PROPERTY P_pParentMzTool : POINTER TO FB_MzBase
GET
END_GET
END_PROPERTY

PROPERTY P_pPiece : POINTER TO FB_PieceBase
GET
P_pPiece := pPiece;
END_GET
SET
pPiece := P_pPiece;
END_SET
END_PROPERTY

PROPERTY P_pXDrive : POINTER TO FB_XYDriveBase
GET
P_pXDrive := pXDrive;
END_GET
END_PROPERTY

PROPERTY P_pYDrive : POINTER TO FB_XYDriveBase
GET
P_pYDrive := pYDrive;
END_GET
END_PROPERTY

PROPERTY P_rToolRadius : REAL
GET
END_GET
END_PROPERTY

PROPERTY P_stAbsPosPhys : ST_3DPoint
GET
END_GET
END_PROPERTY

PROPERTY P_stAbsPosTotal : ST_3DPoint
GET
P_stAbsPosTotal := P_stAbsPosPhys;
END_GET
END_PROPERTY

PROPERTY P_stCurrentPosPhys : ST_3DPoint
GET
END_GET
END_PROPERTY

PROPERTY P_stCurrentPosTotal : ST_3DPoint
GET
P_stCurrentPosTotal := P_stCurrentPosPhys;
END_GET
END_PROPERTY

PROPERTY P_stError : ST_Error
GET
P_stError := stError;
END_GET
END_PROPERTY

PROPERTY P_stOffset : ST_3DPoint
GET
P_stOffset := stOffset;
END_GET
SET
stOffset := P_stOffset;
END_SET
END_PROPERTY

PROPERTY P_stRelPos : ST_3DPoint
GET
P_stRelPos := stRelPos;
END_GET
SET
stRelPos := P_stRelPos;
END_SET
END_PROPERTY

END_FUNCTION_BLOCK

// ---- Objects/FB_SlotList.TcPOU
FUNCTION_BLOCK FB_SlotList
VAR_INPUT
END_VAR
VAR_OUTPUT
END_VAR
VAR
	pHead	: POINTER TO ST_POINTER2;
	pTail	: POINTER TO ST_POINTER2;
	pCurrent: POINTER TO ST_POINTER2;
	nCount	: UINT;
END_VAR

PROPERTY P_nCount : UINT
GET
P_nCount := nCount;
END_GET
END_PROPERTY

METHOD M_GetAtIndex : POINTER TO FB_Slot
VAR_INPUT
	nIndex : UINT;
END_VAR

VAR
	i : UINT;
	pItem : POINTER TO ST_POINTER2;
END_VAR
//mit Index ist die fortlaufende Nummer eines Slots in der Liste gemeint
IF nIndex > 0 AND nIndex <= nCount THEN
	pItem := pHead;
	FOR i := 1 TO nIndex - 1 BY 1 DO
		pItem := pItem^.pNext;
	END_FOR
	M_GetAtIndex := pItem^.pContent;
END_IF
END_METHOD

METHOD M_GetAtNr : POINTER TO FB_Slot
VAR_INPUT
	nNr	: UINT;
END_VAR

VAR
	pPointer : POINTER TO ST_POINTER2;
	pSlot: POINTER TO FB_Slot; 
END_VAR
//Gibt Slot anhand der SlotNr zurück
pPointer := pHead;
WHILE pPointer > 0 DO
	pSlot := pPointer^.pContent;
	IF pSlot^.P_nNr = nNr THEN
		EXIT;
	ELSE
		pSlot := 0;
	END_IF
	pPointer := pPointer^.pNext;
END_WHILE

IF pSlot > 0 THEN
	M_GetAtNr := pSlot;
END_IF
END_METHOD

METHOD M_SetCurrentToHead : BOOL
VAR_INPUT
END_VAR
pCurrent := pHead;
END_METHOD

METHOD M_Add : ERRORID
VAR_INPUT
	pSlot : POINTER TO FB_Slot;
END_VAR

VAR
	pNew : POINTER TO ST_POINTER2;
END_VAR
pNew := pHead;
WHILE pNew > 0 DO
	IF pNew^.pContent = pSlot THEN
		M_Add := 43434;
		RETURN;
	END_IF
	pNew := pNew^.pNext;
END_WHILE

pNew := __NEW(ST_Pointer2);
MEMSET(pNew,0,SIZEOF(ST_POINTER2));
pNew^.pContent := pSlot;
IF pHead = 0 THEN
	pHead := pTail := pNew;
ELSE
	pNew^.pPrev := pTail; 
	pTail^.pNext := pNew;
	pTail := pNew;
END_IF
nCount := nCount + 1;
END_METHOD

METHOD M_Reset
VAR_INPUT
END_VAR

VAR
	pDelete : POINTER TO ST_Pointer2;
	pNext	: POINTER TO ST_Pointer2;
	pSlot	: POINTER TO FB_SLOT;
END_VAR
pDelete := pHead;
WHILE  pDelete > 0 DO
	pNext := pDelete^.pNext;
	pSlot := pDelete^.pContent; 
	IF pSlot > 0 THEN
		__DELETE(pSlot);
	END_IF
	__DELETE(pDelete);
	pDelete := pNext;
END_WHILE
pHead := 0;
pTail := 0;
pCurrent := 0;
nCount := 0;
END_METHOD

METHOD M_GetNext : POINTER TO FB_Slot
VAR_INPUT
END_VAR

VAR
	pSlot : POINTER TO FB_Slot;
END_VAR
IF pCurrent > 0 THEN
	pSlot := pCurrent^.pContent;
	IF pSlot > 0 THEN
		M_GetNext := pSlot;
	END_IF
	pCurrent := pCurrent^.pNext;
END_IF
END_METHOD

END_FUNCTION_BLOCK

// ---- Objects/Targets/Passive/FB_Workplate.TcPOU
FUNCTION_BLOCK FB_Workplate EXTENDS FB_SlotTarget
VAR_INPUT
END_VAR
VAR_OUTPUT
END_VAR
VAR
	rCollHeight			: REAL;
	bCalcCollHeight		: BOOL;
	iter				: FB_ObjCollectIteratorDeep;
	pTarget				: POINTER TO FB_TargetBase;
	stAbsPosCenter		: ST_3DPoint;
	fbRectangle			: FB_Rectangle;
	nParentSlotNr		: UINT;		//Workplate befindet sich zwar an keinem Slot, aber virtuell in der GUI (am Root)
END_VAR

IF bCalcCollHeight THEN
	bCalcCollHeight := FALSE;
	fbRectangle(X1:=0.0, Y1:=0.0, X2:=stDimension.Width, Y2:=stDimension.Depth);
	pTarget := M_GetHighestTarget(fbRectAngle,0.0);
	IF pTarget > 0 THEN
		IF pTarget^.P_rAbsFreeHeight > P_rAbsFreeHeight THEN
			rCollHeight := pTarget^.P_rAbsFreeHeight + 1000.0;
		ELSE
			rCollHeight := P_rAbsFreeHeight + 1000.0;
		END_IF
	ELSE
		rCollHeight := P_rAbsFreeHeight + 1000.0;
	END_IF
END_IF

METHOD FB_init : BOOL
VAR_INPUT
	bInitRetains : BOOL; // if TRUE, the retain variables are initialized (warm start / cold start)
	bInCopyCode : BOOL;  // if TRUE, the instance afterwards gets moved into the copy code (online change)
END_VAR
eObjectType := E_ObjectType.OBJECTTYPE_Workplate;
eObjectGroup := E_ObjectGroup.OBJECTGROUP_Target;
END_METHOD

METHOD M_AddChild : ERRORID
VAR_INPUT
	pObject : POINTER TO FB_Object;
	nSlotNr	: UINT;
	nIndex 	: INT;
END_VAR
//Kann alle Targets aufnehmen
IF pObject > 0 THEN
	IF pObject^.M_bIsGroup(E_ObjectGroup.OBJECTGROUP_Target) THEN
		M_AddChild := SUPER^.M_AddChild(pObject,nSlotNr,nIndex);
	ELSE
		M_AddChild := E_ErrorIdObjMgmt.ERRORID_InvalidParentObject;
	END_IF
ELSE
	M_AddChild := E_ErrorIdObjMgmt.ERRORID_InvalidParentObject;
END_IF
END_METHOD

METHOD M_ClearAllProps
VAR_INPUT
	bIgnoreParent : BOOL; //Es wird das gesamte OD gelöscht. -> Zeiger auf Parent nicht mehr gültig!
END_VAR
SUPER^.M_ClearAllProps(bIgnoreParent);
rCollHeight := 0;
END_METHOD

METHOD M_GetAllProps : ERRORID
VAR_INPUT
	refCmdData : REFERENCE TO  ST_CmdData;
END_VAR
SUPER^.M_GetAllProps(refCmdData);

refCmdData.n32Data[1] := nParentSlotNr;
END_METHOD

METHOD M_SetAllProps : ERRORID
VAR_INPUT
	refCmdData : REFERENCE TO  ST_CmdData;
END_VAR
M_SetAllProps := SUPER^.M_SetAllProps(refCmdData);
IF M_SetAllProps > 0 THEN
	RETURN;
END_IF

nParentSlotNr := DINT_TO_UINT(refCmdData.n32Data[1]);
END_METHOD

PROPERTY P_bCalcCollisHeight : BOOL
SET
bCalcCollHeight := P_bCalcCollisHeight;
END_SET
END_PROPERTY

PROPERTY P_nParentSlotNr : UINT
GET
P_nParentSlotNr := nParentSlotNr;
END_GET
END_PROPERTY

PROPERTY P_rCollHeight : REAL
GET
P_rCollHeight := rCollHeight;
END_GET
SET
rCollHeight := P_rCollHeight;
END_SET
END_PROPERTY

END_FUNCTION_BLOCK

// ---- Objects/Targets/Passive/FB_SlotTarget.TcPOU
FUNCTION_BLOCK FB_SlotTarget EXTENDS FB_TargetBase IMPLEMENTS I_SlotTarget
VAR_INPUT
END_VAR
VAR_OUTPUT
END_VAR
VAR
	fbSlotList			: FB_SlotList;
	nNumberOfSlots		: UINT;
	nFirstSlotPropIndex	: UINT;	//erster Index für Slots (benötigt in M_SetSingleProps)
	nLastSlotPropIndex	: UINT;	//letzte Index für Slots (benötigt in M_SetSingleProps)
END_VAR

SUPER^();

METHOD M_AddChild : ERRORID
VAR_INPUT
	pObject : POINTER TO FB_Object;
	nSlotNr	: UINT;
	nIndex 	: INT;
END_VAR

VAR
	pSlot : POINTER TO FB_Slot;
END_VAR
//In den abgeleiteten Tool-FBs wird überprüft, ob das entsprechende Objekt als Child tauglich ist
IF pObject > 0 THEN
	IF nSlotNr > 0 THEN
		pSlot := fbSlotList.M_GetAtNr(nSlotNr);
		IF pSlot > 0 THEN
			IF pSlot^.P_pChild = 0 THEN
				//Object darf selber noch an keinem Parent hängen
				IF pObject^.P_pParentObject = 0 THEN
					pSlot^.P_pChild := pObject;
					pObject^.P_pObjCollectNode := pObjCollectNode^.nodes.M_AddNewNode(pObject,nIndex);
					pObject^.M_UpdateParent();
				ELSE
					M_AddChild := E_ErrorIdObjMgmt.ERRORID_ObjectAlreadyOnAnotherParent;
				END_IF
			ELSE //Slot bereits belegt
				M_AddChild := E_ErrorIdObjMgmt.ERRORID_SlotIsAlreadyOccupied;
			END_IF		
		ELSE
			M_AddChild := E_ErrorIdObjMgmt.ERRORID_InvalidSlotNumber;			
		END_IF	
	ELSE
		M_AddChild := SUPER^.M_AddChild(pObject,nSlotNr,nIndex);
	END_IF
ELSE
	M_AddChild := E_ErrorIdObjMgmt.ERRORID_InvalidParentObject;
END_IF
END_METHOD

METHOD M_ApplyPos : ERRORID
VAR_INPUT
	eTargetRef 		: E_TargetRef;
	nPointSlotNr	: UINT;
	stPos 			: ST_3DPoint;
	bXPos			: BOOL;
	bYPos			: BOOL;
	bZPos			: BOOL;	
END_VAR

VAR
	stAbsPos		: ST_3DPoint;
	pSlot			: POINTER TO FB_Slot;
END_VAR
IF eTargetRef = E_TargetRef.TARGETREF_Slot THEN
	stAbsPos := P_stAbsPosLB;
	pSlot := M_GetSlot(nPointSlotNr);
	IF pSlot > 0 THEN
		IF bXPos THEN
			pSlot^.P_rRelPosX := stPos.X - stAbsPos.X;
		END_IF
		IF bYPos THEN
			pSlot^.P_rRelPosY := stPos.Y - stAbsPos.Y;
		END_IF
		IF bZPos THEN
			pSlot^.P_rRelPosZ := stPos.Z - stAbsPos.Z;
			P_pWorkplate^.P_bCalcCollisHeight := TRUE;
		END_IF
	ELSE
		M_ApplyPos := E_ErrorIdCmd.ERRORID_InvalidTargetSlot;
	END_IF
ELSE
	M_ApplyPos := SUPER^.M_ApplyPos(eTargetRef, nPointSlotNr, stPos,bXPos, bYPos, bZPos);	
END_IF
END_METHOD

METHOD M_ClearAllProps
VAR_INPUT
	bIgnoreParent : BOOL; //Es wird das gesamte OD gelöscht. -> Zeiger auf Parent nicht mehr gültig!
END_VAR
fbSlotList.M_Reset();
SUPER^.M_ClearAllProps(bIgnoreParent);
END_METHOD

METHOD M_GetAbsPos : ST_3DPoint
VAR_INPUT
	pChildPos	: POINTER TO ST_3DPoint;
	eTargetRef 	: E_TargetRef;
	nParam1		: UINT;
 	nParam2		: UINT;
	nParam3		: USINT;
	nParam4		: USINT;
	nZLevel		: USINT;
END_VAR
VAR_OUTPUT
	nErrorId 	: ERRORID;
	lrAngle		: LREAL;
END_VAR
VAR
	stLocPos : ST_3DPoint;
	pSlot : POINTER TO FB_Slot;
END_VAR
IF eTargetRef = E_TargetRef.TARGETREF_Slot THEN
	//Slotnummer checken
	pSlot := M_GetSlot(nParam1);
	IF pSlot > 0 THEN
		stLocPos := F_Add3DPoints(pSlot^.P_stRelPos,stRelPos);
		stLocPos.Z := stLocPos.Z + stDimension.Height;
		//kann es mal sein, dass hier das ParentTarget = 0 ist?
		//ja -> bei der Workplate
		IF pChildPos > 0 THEN
			stLocPos := F_Add3DPoints(stLocPos,pChildPos^);
		END_IF
		IF pParentTarget > 0 THEN
			IF pParentSlot > 0 THEN
				M_GetAbsPos := pParentTarget^.M_GetAbsPos(pChildPos := ADR(stLocPos), eTargetRef:= E_TargetRef.TARGETREF_Slot,
															nParam1:= pParentSlot^.P_nNr,
															nParam2:= 0, nParam3:= 0, nParam4:= 0,nZLevel:= 0, lrAngle=> lrAngle,
															nErrorId=> nErrorId);		
			ELSE
				M_GetAbsPos := pParentTarget^.M_GetAbsPos(pChildPos := ADR(stLocPos), eTargetRef:= E_TargetRef.TARGETREF_LeftBottom,
																nParam1:= 0,
																nParam2:= 0, nParam3:= 0, nParam4:= 0, nZLevel:= 0,
																lrAngle => lrAngle, nErrorId=> nErrorId);
			END_IF
		ELSE
			M_GetAbsPos := stLocPos;
		END_IF		
	ELSE
		nErrorId := E_ErrorIdCmd.ERRORID_InvalidTargetSlot;
	END_IF
	
ELSE
	M_GetAbsPos := SUPER^.M_GetAbsPos(pChildPos := pChildPos, eTargetRef:= eTargetRef,
													nParam1:= nParam1,
													nParam2:= nParam2, nParam3:= nParam3, nParam4:= 0, nZLevel:= nZLevel,
													lrAngle => lrAngle, nErrorId=> nErrorId);	
END_IF
END_METHOD

METHOD M_GetAllProps : ERRORID
VAR_INPUT
	refCmdData : REFERENCE TO  ST_CmdData;
END_VAR

VAR
	i : UINT;
	pSlot		: POINTER TO FB_Slot;
	pPieceSlot	: POINTER TO FB_PieceSlot;
END_VAR
SUPER^.M_GetAllProps(refCmdData);

nCurrentPropIndex := nCurrentPropIndex + 1;

refCmdData.n32Data[nCurrentPropIndex] := fbSlotList.P_nCount;

fbSlotList.M_SetCurrentToHead();

IF (eObjectGroup AND E_ObjectGroup.OBJECTGROUP_Rack) = E_ObjectGroup.OBJECTGROUP_Rack THEN
	FOR i := 1 TO fbSlotList.P_nCount BY 1 DO
		pPieceSlot := fbSlotList.M_GetNext();
		IF pPieceSlot > 0 THEN
			nCurrentPropIndex := nCurrentPropIndex + 1;
			refCmdData.n32Data[nCurrentPropIndex] := pPieceSlot^.P_nNr;
			nCurrentPropIndex := nCurrentPropIndex + 1;
			refCmdData.n32Data[nCurrentPropIndex] := REAL_TO_DINT(pPieceSlot^.P_rRelPosX);
			nCurrentPropIndex := nCurrentPropIndex + 1;
			refCmdData.n32Data[nCurrentPropIndex] := REAL_TO_DINT(pPieceSlot^.P_rRelPosY);
			nCurrentPropIndex := nCurrentPropIndex + 1;
			refCmdData.n32Data[nCurrentPropIndex] := REAL_TO_DINT(pPieceSlot^.P_rRelPosZ);
			nCurrentPropIndex := nCurrentPropIndex + 1;
			refCmdData.n32Data[nCurrentPropIndex] := REAL_TO_DINT(pPieceSlot^.P_rDepth);
		END_IF		
	END_FOR	
ELSE
	FOR i := 1 TO fbSlotList.P_nCount BY 1 DO
		pSlot := fbSlotList.M_GetNext();
		IF pSlot > 0 THEN
			nCurrentPropIndex := nCurrentPropIndex + 1;
			refCmdData.n32Data[nCurrentPropIndex] := pSlot^.P_nNr;
			nCurrentPropIndex := nCurrentPropIndex + 1;
			refCmdData.n32Data[nCurrentPropIndex] := REAL_TO_DINT(pSlot^.P_rRelPosX);
			nCurrentPropIndex := nCurrentPropIndex + 1;
			refCmdData.n32Data[nCurrentPropIndex] := REAL_TO_DINT(pSlot^.P_rRelPosY);
			nCurrentPropIndex := nCurrentPropIndex + 1;
			refCmdData.n32Data[nCurrentPropIndex] := REAL_TO_DINT(pSlot^.P_rRelPosZ);
		END_IF		
	END_FOR	
END_IF
END_METHOD

METHOD M_GetSlot : POINTER TO FB_Slot
VAR_INPUT
	nSlotNr : UINT;
END_VAR
M_GetSlot := fbSlotList.M_GetAtNr(nSlotNr);
END_METHOD

METHOD M_GetSlotFromChild : POINTER TO FB_Slot
VAR_INPUT
	pObject : POINTER TO FB_Object;
END_VAR

VAR
	pSlot : POINTER TO FB_Slot;
END_VAR
//Die SlotList iterieren und vergleichen ob Objekte übereinstimmen
fbSlotList.M_SetCurrentToHead();
REPEAT
	pSlot := fbSlotList.M_GetNext();
	IF pSlot > 0 THEN
		IF pSlot^.P_pChild = pObject THEN
			M_GetSlotFromChild := pSlot;
			EXIT;
		END_IF
	END_IF
UNTIL pSlot = 0
END_REPEAT
END_METHOD

METHOD M_SetAllProps : ERRORID
VAR_INPUT
	refCmdData : REFERENCE TO  ST_CmdData;
END_VAR

VAR
	i : UINT;
	pSlot 		: POINTER TO FB_Slot;
	pPieceSlot	: POINTER TO FB_PieceSlot;
END_VAR
M_SetAllProps := SUPER^.M_SetAllProps(refCmdData);

IF M_SetAllProps > 0 THEN
	RETURN;
END_IF

//Slots parametrieren
nCurrentPropIndex := nCurrentPropIndex + 1;
nFirstSlotPropIndex := nCurrentPropIndex;
nNumberOfSlots := DINT_TO_UINT(refCmdData.n32Data[nCurrentPropIndex]);

//Falls SlotList noch nicht existiert, dann neue erstellen
IF fbSlotList.P_nCount = 0 THEN
	FOR i:= 1 TO nNumberOfSlots BY 1 DO
		IF (eObjectGroup AND E_ObjectGroup.OBJECTGROUP_Rack) = E_ObjectGroup.OBJECTGROUP_Rack THEN
			pPieceSlot := __NEW(FB_PieceSlot(pOwner := THIS));
			pSlot := pPieceSlot;
		ELSE
			pSlot := __NEW(FB_Slot(pOwner := THIS));
		END_IF
		
		fbSlotList.M_Add(pSlot);
		nCurrentPropIndex := nCurrentPropIndex + 1;
		pSlot^.P_nNr := DINT_TO_USINT(refCmdData.n32Data[nCurrentPropIndex]);
		nCurrentPropIndex := nCurrentPropIndex + 1;
		pSlot^.P_rRelPosX := DINT_TO_REAL(refCmdData.n32Data[nCurrentPropIndex]);
		nCurrentPropIndex := nCurrentPropIndex + 1;
		pSlot^.P_rRelPosY := DINT_TO_REAL(refCmdData.n32Data[nCurrentPropIndex]);
		nCurrentPropIndex := nCurrentPropIndex + 1;
		pSlot^.P_rRelPosZ := DINT_TO_REAL(refCmdData.n32Data[nCurrentPropIndex]);
		
		IF (eObjectGroup AND E_ObjectGroup.OBJECTGROUP_Rack) = E_ObjectGroup.OBJECTGROUP_Rack THEN
			nCurrentPropIndex := nCurrentPropIndex + 1;
			pPieceSlot^.P_rDepth := DINT_TO_REAL(refCmdData.n32Data[nCurrentPropIndex]);
		END_IF
	END_FOR
ELSE
	IF nNumberOfSlots <> fbSlotList.P_nCount THEN	//Anzahl der Slots dürfen sich nicht ändern
		M_SetAllProps := E_ErrorIdObjMgmt.ERRORID_ChangeNoOfSlotsNotAllowed;
		RETURN;		
	END_IF

	FOR i:= 1 TO nNumberOfSlots BY 1 DO
		nCurrentPropIndex := nCurrentPropIndex + 1;
		IF (eObjectGroup AND E_ObjectGroup.OBJECTGROUP_Rack) = E_ObjectGroup.OBJECTGROUP_Rack THEN
			pPieceSlot := fbSlotList.M_GetAtNr(DINT_TO_USINT(refCmdData.n32Data[nCurrentPropIndex]));
			IF pPieceSlot > 0 THEN
				nCurrentPropIndex := nCurrentPropIndex + 1;
				pPieceSlot^.P_rRelPosX := DINT_TO_REAL(refCmdData.n32Data[nCurrentPropIndex]);
				nCurrentPropIndex := nCurrentPropIndex + 1;
				pPieceSlot^.P_rRelPosY := DINT_TO_REAL(refCmdData.n32Data[nCurrentPropIndex]);
				nCurrentPropIndex := nCurrentPropIndex + 1;
				pPieceSlot^.P_rRelPosZ := DINT_TO_REAL(refCmdData.n32Data[nCurrentPropIndex]);
				nCurrentPropIndex := nCurrentPropIndex + 1;
				pPieceSlot^.P_rDepth := DINT_TO_REAL(refCmdData.n32Data[nCurrentPropIndex]);
			ELSE
				M_SetAllProps := 222;
				RETURN;
			END_IF 
		ELSE
			pSlot := fbSlotList.M_GetAtNr(DINT_TO_USINT(refCmdData.n32Data[nCurrentPropIndex]));
			IF pSlot > 0 THEN
				nCurrentPropIndex := nCurrentPropIndex + 1;
				pSlot^.P_rRelPosX := DINT_TO_REAL(refCmdData.n32Data[nCurrentPropIndex]);
				nCurrentPropIndex := nCurrentPropIndex + 1;
				pSlot^.P_rRelPosY := DINT_TO_REAL(refCmdData.n32Data[nCurrentPropIndex]);
				nCurrentPropIndex := nCurrentPropIndex + 1;
				pSlot^.P_rRelPosZ := DINT_TO_REAL(refCmdData.n32Data[nCurrentPropIndex]);
			ELSE
				M_SetAllProps := 222;
				RETURN;
			END_IF	
		END_IF
	END_FOR
END_IF
nLastSlotPropIndex := nCurrentPropIndex;
nNoOfProps := nCurrentPropIndex + 1;
END_METHOD

METHOD M_SetSingleProp : ERRORID
VAR_INPUT
	refCmdData : REFERENCE TO  ST_CmdData;
END_VAR

VAR
	nSlotNr		: UINT;
	nIndex		: UINT;
	pSlot		: POINTER TO FB_Slot;
	pPieceSlot	: POINTER TO FB_PieceSlot;
END_VAR
//Handelt es sich bei dem PropNr um eine SlotPropNr?
IF refCmdData.aHeader[1] >= nFirstSlotPropIndex AND refCmdData.aHeader[1] <= nLastSlotPropIndex THEN
	nIndex := (refCmdData.aHeader[1]- nFirstSlotPropIndex);
	//Beachten normale Slots oder PieceSlots
	IF (eObjectGroup AND E_ObjectGroup.OBJECTGROUP_Rack) = E_ObjectGroup.OBJECTGROUP_Rack THEN //PieceSlots
		IF nIndex MOD 5 = 0 THEN
			nSlotNr := nIndex / 5;
		ELSE
			nSlotNr := nIndex / 5 + 1;
		END_IF
		pPieceSlot := fbSlotList.M_GetAtNr(nSlotNr);
		IF pPieceSlot > 0 THEN
			nIndex := nIndex - ((nSlotNr - 1)* 5);
			CASE nIndex OF
				2:	pPieceSlot^.P_rRelPosX := DINT_TO_REAL(refCmdData.n32Data[0]);
				
				3:	pPieceSlot^.P_rRelPosY := DINT_TO_REAL(refCmdData.n32Data[0]);
				
				4:	pPieceSlot^.P_rRelPosZ := DINT_TO_REAL(refCmdData.n32Data[0]);
					P_pWorkplate^.P_bCalcCollisHeight := TRUE;
				
				5:	pPieceSlot^.P_rDepth := DINT_TO_REAL(refCmdData.n32Data[0]);
			END_CASE
		END_IF
	ELSE //normale Slots
		IF nIndex MOD 4 = 0 THEN
			nSlotNr := nIndex / 4;
		ELSE
			nSlotNr := nIndex / 4 + 1;
		END_IF
		pSlot := fbSlotList.M_GetAtNr(nSlotNr);
		IF pSlot > 0 THEN
			nIndex := nIndex - ((nSlotNr - 1)* 4);
			CASE nIndex OF
				2:	pSlot^.P_rRelPosX := DINT_TO_REAL(refCmdData.n32Data[0]);
				
				3:	pSlot^.P_rRelPosY := DINT_TO_REAL(refCmdData.n32Data[0]);
				
				4:	pSlot^.P_rRelPosZ := DINT_TO_REAL(refCmdData.n32Data[0]);
					P_pWorkplate^.P_bCalcCollisHeight := TRUE;
			END_CASE
		END_IF	
	END_IF
ELSE
	M_SetSingleProp := SUPER^.M_SetSingleProp(refCmdData);
END_IF
END_METHOD

END_FUNCTION_BLOCK

// ---- Functions/F_Add3DPoints.TcPOU
FUNCTION F_Add3DPoints : ST_3DPoint
VAR_INPUT
	stPoint1	: ST_3DPoint;
	stPoint2	: ST_3DPoint;
END_VAR
VAR
	_stPoint	: ST_3DPoint;
END_VAR

_stPoint.X := stPoint1.X + stPoint2.X;
_stPoint.Y := stPoint1.Y + stPoint2.Y;
_stPoint.Z := stPoint1.Z + stPoint2.Z;
F_Add3DPoints := _stPoint;

END_FUNCTION

// ---- Objects/FB_PieceSlot.TcPOU
{attribute 'enable_dynamic_creation'}
FUNCTION_BLOCK FB_PieceSlot EXTENDS FB_Slot
VAR_INPUT
END_VAR
VAR_OUTPUT
END_VAR
VAR
	rDepth	 : REAL;
END_VAR

PROPERTY P_rDepth : REAL
GET
P_rDepth := rDepth;
END_GET
SET
rDepth := P_rDepth;
END_SET
END_PROPERTY

PROPERTY P_pPiece : POINTER TO FB_PieceBase
GET
IF pChild > 0 THEN
	P_pPiece := pChild;
END_IF
END_GET
SET
IF P_pPiece > 0 THEN
	pChild := P_pPiece;
ELSE
	pChild := 0;	
END_IF
END_SET
END_PROPERTY

END_FUNCTION_BLOCK

// ---- Objects/Pieces/FB_PieceBase.TcPOU
FUNCTION_BLOCK FB_PieceBase EXTENDS FB_Object
VAR_INPUT
END_VAR
VAR_OUTPUT
	bUsingPiece			: BOOL;	
END_VAR
VAR
	pParentObject		: POINTER TO FB_Object;
	stDimension			: ST_3DDimension;
	rSlotDiameter		: REAL;
	stOffset			: ST_3DPoint;	//Offset
	rZOverlapTool		: REAL;
	rZOverlapSlot		: REAL;
	rMeasureDistance	: REAL;
	rDockOffset			: REAL;
	nCurrentPropIndex	: USINT;
	nSpecPropIndex		: USINT;			//erster Index für Specialproperties
	bIgnoreOffset		: BOOL;
END_VAR

METHOD M_UpdateParent
VAR_INPUT
END_VAR
IF pObjCollectNode > 0 AND_THEN pObjCollectNode^.pOwnerColl > 0 THEN
	pParentObject := pObjCollectNode^.pOwnerColl^.pOwnerNode^.P_pObject;
ELSE
	pParentObject := 0;
END_IF

IF pParentObject > 0 THEN
	pParentSlot := pParentObject^.M_GetSlotFromChild(THIS);
ELSE
	pParentSlot := 0;
END_IF
END_METHOD

METHOD M_GetPropCheckSum : UINT
VAR_INPUT
END_VAR

VAR
	stData 		: ST_CmdData;
END_VAR
M_GetAllProps(stData);
wChecksum := F_DATA_TO_CRC16_CCITT(ADR(stData.n32Data[0]),nNoOfProps * 4,16#FFFF);
M_GetPropCheckSum := wChecksum;
END_METHOD

PROPERTY P_stDimension : ST_3DDimension
GET
P_stDimension := stDimension;
END_GET
END_PROPERTY

PROPERTY P_rDockOffset : REAL
GET
P_rDockOffset := rDockOffset;
END_GET
END_PROPERTY

{attribute 'object_name' := 'M_CheckProps'}
METHOD M_CheckProps : ERRORID
END_METHOD

PROPERTY P_rZOverlapSlot : REAL
GET
P_rZOverlapSlot := rZOverlapSlot;
END_GET
END_PROPERTY

PROPERTY P_pLatestChild : POINTER TO FB_PieceBase
GET
P_pLatestChild := THIS;
END_GET
END_PROPERTY

PROPERTY P_rZOverlapTool : REAL
GET
P_rZOverlapTool := rZOverlapTool;
END_GET
END_PROPERTY

PROPERTY P_stOffset : ST_3DPoint
GET
P_stOffset := stOffset;
END_GET
SET
stOffset := P_stOffset;
END_SET
END_PROPERTY

{attribute 'object_name' := 'M_ClearAllProps'}
METHOD M_ClearAllProps

VAR_INPUT
	bIgnoreParent : BOOL; //Es wird das gesamte OD gelöscht. -> Zeiger auf Parent nicht mehr gültig!
END_VAR
IF NOT bIgnoreParent THEN
	IF pParentSlot > 0 THEN
		pParentSlot^.P_pChild := 0;
	END_IF	
END_IF
nObjectID := 0;
pParentObject := 0;
pParentSlot := 0;
pObjCollectNode := 0;
END_METHOD

METHOD M_GetRelPosTopCenter : ST_3DPoint
VAR_INPUT
END_VAR
VAR
	stPosTemp : ST_3DPoint;
	pPieceSlot : POINTER TO FB_PieceSlot;
END_VAR
IF pParentObject > 0 THEN
	IF pParentObject^.M_bIsGroup(E_ObjectGroup.OBJECTGROUP_Target) THEN
		IF pParentSlot > 0 THEN
			pPieceSlot := pParentSlot;
			stPosTemp := pPieceSlot^.P_stRelPos;
			//Wenn OverlapSlot > SlotTiefe, dann sitzt Piece auf dem Grund des Slots auf
			IF rZOverlapSlot > pPieceSlot^.rDepth THEN
				stPosTemp.Z := stPosTemp.Z - pPieceSlot^.rDepth + stDimension.Height;
			ELSE
				stPosTemp.Z := stPosTemp.Z - rZOverlapSlot + stDimension.Height;
			END_IF
			IF bIgnoreOffset THEN
				M_GetRelPosTopCenter := stPosTemp;
			ELSE
				M_GetRelPosTopCenter := F_Add3DPoints(stPosTemp,stOffset);	
			END_IF
		END_IF
	END_IF
END_IF
END_METHOD

{attribute 'object_name' := 'M_SetSingleProp'}
METHOD M_SetSingleProp : ERRORID
VAR_INPUT
	refCmdData	: REFERENCE TO ST_CmdData;
END_VAR
CASE refCmdData.aHeader[1] OF
	0,1:
		M_SetSingleProp := E_ErrorIdCmd.ERRORID_InvalidProperty;
	2:	stDimension.Width := DINT_TO_REAL(refCmdData.n32Data[0]);
	3:	stDimension.Depth := DINT_TO_REAL(refCmdData.n32Data[0]);
	4:	stDimension.Height := DINT_TO_REAL(refCmdData.n32Data[0]);
	5:	rSlotDiameter := DINT_TO_REAL(refCmdData.n32Data[0]);
	6:	rZOverlapTool := DINT_TO_REAL(refCmdData.n32Data[0]);
	7:	rZOverlapSlot := DINT_TO_REAL(refCmdData.n32Data[0]);
	8:	stOffset.X := DINT_TO_REAL(refCmdData.n32Data[0]);
	9:	stOffset.Y := DINT_TO_REAL(refCmdData.n32Data[0]);
	10:	stOffset.Z := DINT_TO_REAL(refCmdData.n32Data[0]);
	11: rMeasureDistance := DINT_TO_REAL(refCmdData.n32Data[0]);
	12:	rDockOffset := DINT_TO_REAL(refCmdData.n32Data[0]);
END_CASE
END_METHOD

METHOD M_ClearOffset
VAR_INPUT
END_VAR
stOffset.X := 0.0;
stOffset.Y := 0.0;
stOffset.Z := 0.0;
END_METHOD

PROPERTY P_rMeasureDistance : REAL
GET
P_rMeasureDistance := rMeasureDistance;
END_GET
END_PROPERTY

{attribute 'object_name' := 'M_GetAllProps'}
METHOD M_GetAllProps : ERRORID
VAR_INPUT
	refCmdData	: REFERENCE TO ST_CmdData;
END_VAR
refCmdData.aHeader[0] := nObjectID;
refCmdData.aHeader[1] := eObjectType;
refCmdData.aHeader[2] := 0;

IF pParentObject > 0 THEN
	refCmdData.n32Data[0] := pParentObject^.P_nObjectID;
ELSE
	refCmdData.n32Data[0] := 0;
END_IF

IF pParentSlot > 0 THEN
	refCmdData.n32Data[1] := pParentSlot^.nNr;
ELSE
	refCmdData.n32Data[1] := 0;
END_IF

//Dimensionen lesen
refCmdData.n32Data[2] := REAL_TO_DINT(stDimension.Width);
refCmdData.n32Data[3] := REAL_TO_DINT(stDimension.Depth);
refCmdData.n32Data[4] := REAL_TO_DINT(stDimension.Height);
refCmdData.n32Data[5] := REAL_TO_DINT(rSlotDiameter);
refCmdData.n32Data[6] := REAL_TO_DINT(rZOverlapTool);
refCmdData.n32Data[7] := REAL_TO_DINT(rZOverlapSlot);
refCmdData.n32Data[8] := REAL_TO_DINT(stOffset.X);
refCmdData.n32Data[9] := REAL_TO_DINT(stOffset.Y);
refCmdData.n32Data[10] := REAL_TO_DINT(stOffset.Z);
refCmdData.n32Data[11] := REAL_TO_DINT(rMeasureDistance);
refCmdData.n32Data[12] := REAL_TO_DINT(rDockOffset);
nCurrentPropIndex := 12;
END_METHOD

METHOD M_AddChild : ERRORID
VAR_INPUT
	pObject	: POINTER TO FB_Object;
	nSlotNr	: UINT;
	nIndex 	: INT;
END_VAR
//Pieces könnnen keine Childs aufnehmen
M_AddChild := E_ErrorIdObjMgmt.ERRORID_ObjectCanNotTakeChilds;
END_METHOD

{attribute 'object_name' := 'M_SetAllProps'}
METHOD M_SetAllProps : ERRORID
VAR_INPUT
	refCmdData	: REFERENCE TO ST_CmdData;
END_VAR
IF fbObjectDirectory.M_GetObjPointer(DINT_TO_UINT(refCmdData.n32Data[0])) = 0 THEN
	M_SetAllProps := E_ErrorIdObjMgmt.ERRORID_InvalidParentObject;
	RETURN;
END_IF

//ParentSlot unterschiedlich?

(*IF pParentSlot = 0 THEN
	M_SetAllProps := M_SetParent(aI_Object[refCmdData.n32Data[0]],DINT_TO_UINT(refCmdData.n32Data[1]));
ELSE
	IF pParentSlot^.P_nNr <> DINT_TO_UINT(refCmdData.n32Data[1]) THEN
		M_SetAllProps := M_SetParent(aI_Object[refCmdData.n32Data[0]],DINT_TO_UINT(refCmdData.n32Data[1]));
	END_IF
END_IF

IF M_SetAllProps > 0 THEN
	RETURN;
END_IF*)

//Dimensionen setzen
stDimension.Width := DINT_TO_REAL(refCmdData.n32Data[2]);
stDimension.Depth := DINT_TO_REAL(refCmdData.n32Data[3]);
stDimension.Height := DINT_TO_REAL(refCmdData.n32Data[4]);
rSlotDiameter := DINT_TO_REAL(refCmdData.n32Data[5]);
rZOverlapTool := DINT_TO_REAL(refCmdData.n32Data[6]);
rZOverlapSlot := DINT_TO_REAL(refCmdData.n32Data[7]);
stOffset.X := DINT_TO_REAL(refCmdData.n32Data[8]);
stOffset.Y := DINT_TO_REAL(refCmdData.n32Data[9]);
stOffset.Z := DINT_TO_REAL(refCmdData.n32Data[10]);
rMeasureDistance := DINT_TO_REAL(refCmdData.n32Data[11]);
rDockOffset := DINT_TO_REAL(refCmdData.n32Data[12]);
nCurrentPropIndex := 12;
nNoOfProps := nCurrentPropIndex + 1;
END_METHOD

PROPERTY P_nCntSlots : UINT
GET
END_GET
END_PROPERTY

PROPERTY P_bIgnoreOffset : BOOL
SET
bIgnoreOffset := P_bIgnoreOffset;
END_SET
GET
P_bIgnoreOffset := bIgnoreOffset;
END_GET
END_PROPERTY

END_FUNCTION_BLOCK

// ---- DUTs/Structs/FB_Rectangle.TcPOU
FUNCTION_BLOCK FB_Rectangle
VAR_INPUT
	X1,Y1,X2,Y2 : REAL;	
END_VAR
VAR_OUTPUT
END_VAR
VAR
END_VAR

PROPERTY P_LineLeft : ST_Line
GET
P_LineLeft.X1 := X1;
P_LineLeft.Y1 := Y1;
P_LineLeft.X2 := X1;
P_LineLeft.Y2 := Y2;
END_GET
END_PROPERTY

PROPERTY P_LineRight : ST_Line
GET
P_LineRight.X1 := X2;
P_LineRight.Y1 := Y1;
P_LineRight.X2 := X2;
P_LineRight.Y2 := Y2;
END_GET
END_PROPERTY

METHOD M_Clear
VAR_INPUT
END_VAR
X1 := 0;
Y1 := 0;
X2 := 0;
Y2 := 0;
END_METHOD

PROPERTY P_LineTop : ST_Line
GET
P_LineTop.X1 := X1;
P_LineTop.Y1 := Y2;
P_LineTop.X2 := X2;
P_LineTop.Y2 := Y2;
END_GET
END_PROPERTY

PROPERTY P_LineBottom : ST_Line
GET
P_LineBottom.X1 := X1;
P_LineBottom.Y1 := Y1;
P_LineBottom.X2 := X2;
P_LineBottom.Y2 := Y1;
END_GET
END_PROPERTY

END_FUNCTION_BLOCK

// ---- Hardware/MultiZ/FB_ZM_Home.TcPOU
FUNCTION_BLOCK FB_ZM_Home
VAR_INPUT
	bExecute		: BOOL;
	pFbZAxisRef		: POINTER TO FB_ZAxisRef;
	bMoveToHome		: BOOL;
END_VAR
VAR_OUTPUT
	bBusy		: BOOL;
	bError		: BOOL;
	nErrorId	: ERRORID;
END_VAR
VAR
	fbSdoWrite	: FB_SDO_WRITE;
	nState		: USINT;
	timeOut		: TON;
	bTest		: BOOL;
	tTime		: TIME;
	nErrorState : USINT;
END_VAR

IF bExecute THEN
	IF pFbZAxisRef = 0 THEN
		RETURN;
	END_IF
	
	//Fehler-Simualation
	(*IF pFbZAxisRef^.nChannel = 4 THEN
		bBusy := FALSE;
		bError := TRUE;
		nState := 99;	//go in errorstate
		RETURN;
	END_IF*)
	
	IF pFbZAxisRef^.stInput.nStatus.3 THEN //Error
		pFbZAxisRef^.stStatus.bError := TRUE;
		pFbZAxisRef^.stStatus.bIsMoving := FALSE;
		pFbZAxisRef^.stStatus.bIsHoming := FALSE;
		pFbZAxisRef^.stOutput.nMode := 0;
		pFbZAxisRef^.stOutput.nCtrl := 0;
		nErrorID := F_MultiZError_TO_ErrorId(pFbZAxisRef^.stInput.nError);
		timeOut(IN:= FALSE);
		bBusy := FALSE;
		bError := TRUE;
		nState := 99;	//go in errorstate
		RETURN;
	END_IF
	
	timeOut();
	IF timeOut.Q THEN
		tTime := timeOut.ET;
		nErrorState := nState;
		timeOut(IN:= FALSE);
		pFbZAxisRef^.stStatus.bError := TRUE;
		pFbZAxisRef^.stStatus.bIsMoving := FALSE;
		pFbZAxisRef^.stStatus.bIsHoming := FALSE;
		pFbZAxisRef^.stOutput.nMode := 0;
		pFbZAxisRef^.stOutput.nCtrl := 0;
		CASE nState OF
			0:	//Timeout reset error
				nErrorId := E_ErrorIdMultiZ.ERRORID_ToResetErr;
			3,6: //Timeout wait for setpointacknowledge
				nErrorId := E_ErrorIdMultiZ.ERRORID_ToWaitSetPointAck;
				bTest := TRUE;
			4: //Timeout wait for targetreached
				nErrorId := E_ErrorIdMultiZ.ERRORID_ToWaitTrgtReached;
		ELSE
			nErrorId := E_ErrorIdMultiZ.ERRORID_UnknownError;	
		END_CASE
		bBusy := FALSE;
		bError := TRUE;
		nState := 99;	//go in errorstate
		RETURN;
	END_IF
	
	CASE nState OF
		0:	bBusy := TRUE;
			pFbZAxisRef^.stStatus.bError := FALSE;
			pFbZAxisRef^.stStatus.bIsHomed := FALSE;
			pFbZAxisRef^.stStatus.bIsHoming := TRUE;
			
			//Das zurücksetzen von Fehlern sollte ausschließlich im FB_MultiZRef stattfinden!!!
			//Hier nur abfragen, ob "pFbZAxisRef^.stStatus.bError" und dann in Error gehen	
			IF pFbZAxisRef^.stInput.nStatus.3 THEN //Error
				pFbZAxisRef^.stOutput.nCtrl := 8;	//Error zurücksetzen
				pFbZAxisRef^.stOutput.nVelo := 0;	//Geschwindigkeit auf 0 setzen
				timeOut(IN:= TRUE, PT:=T#1000MS);	//Timer für Timeout starten
			ELSE
				//Mode of Operation setzen
				IF pFbZAxisRef^.P_bInvertInitDir THEN
					pFbZAxisRef^.stOutput.nMode := 7;
				ELSE
					pFbZAxisRef^.stOutput.nMode := 6;
					pFbZAxisRef^.stOutput.nVelo := 50000;
				END_IF
				
				fbSdoWrite(sADSNetID:= pFbZAxisRef^.pMultiZRef^.P_sAdsNetId, nPortNr:= pFbZAxisRef^.pMultiZRef^.P_nAdsPort,
							nIndex:= cRefPos.nIndex, nSubIndex:= pFbZAxisRef^.nChannel, 
							nDataLength:= cRefPos.nLength, nData:= REAL_TO_DINT(pFbZAxisRef^.P_rRefPos) , bExecute:= TRUE);
				nState := 1;
				timeOut(IN:= FALSE);
			END_IF
			
		1:	//Geschwindigkeit setzen
			fbSdoWrite();
			IF NOT fbSdoWrite.bBusy THEN
				IF fbSdoWrite.bError THEN
					nErrorId := fbSdoWrite.nAdsErrorId;
					bBusy := FALSE;
					bError := TRUE;
					nState := 99;	//go in errorstate
				ELSE
					nState := 200;	
				END_IF
				fbSdoWrite(bExecute:= FALSE);
			END_IF
			
		200:
			nState := 201;
			
		201:
			nState := 2;
						
		2:	//Fahrauftrag starten
			pFbZAxisRef^.stOutput.nCtrl := 1;
			pFbZAxisRef^.stStatus.bIsMoving := TRUE;
			timeOut(IN:= TRUE, PT:=T#2000MS);	//Timer für Timeout starten
			nState := 3;
	
		3:	//SetpointAcknowledge?
			IF pFbZAxisRef^.stInput.nStatus.1 THEN
				pFbZAxisRef^.stOutput.nCtrl := 0;	//Fahrauftrag zurücksetzen
				timeOut(IN:= FALSE);
				nState := 4;
			END_IF
			
		4:	//TargetReached?
			IF pFbZAxisRef^.stInput.nStatus.0 THEN
				pFbZAxisRef^.stStatus.bIsMoving := FALSE;	
				pFbZAxisRef^.stOutput.nMode := 1;		//in Positioniermodus umschalten
				timeOut(IN:= FALSE);
				IF bMoveToHome THEN
					pFbZAxisRef^.P_rAbsTargetPos := pFbZAxisRef^.P_rHomePos;
					nState := 5;
				ELSE
					nState := 8;
				END_IF
			ELSE
				timeOut(IN:= TRUE, PT:=T#5S);	//Timer für Timeout starten
			END_IF
			
		5:	//auf HomePos fahren
			pFbZAxisRef^.stOutput.nCtrl := 1;
			pFbZAxisRef^.stStatus.bIsMoving := TRUE;
			timeOut(IN:= TRUE, PT:=T#500MS);	//Timer für Timeout starten
			nState := 6;
			
		6:	//SetpointAcknowledge?
			IF pFbZAxisRef^.stInput.nStatus.1 THEN
				pFbZAxisRef^.stOutput.nCtrl := 0;	//Fahrauftrag zurücksetzen
				timeOut(IN:= FALSE);
				nState := 7;
			END_IF			
			
		7:	//TargetReached?
			IF pFbZAxisRef^.stInput.nStatus.0 THEN
				pFbZAxisRef^.stStatus.bIsMoving := FALSE;
				timeOut(IN:= FALSE);
				nState := 8;
			ELSE
				timeOut(IN:= TRUE, PT:=T#3S);	//Timer für Timeout starten
			END_IF	
		
		8:	IF pFbZAxisRef^.stInput.nStatus.3 THEN		//Error ist in Achse aufgetreten
				pFbZAxisRef^.stStatus.bError := TRUE;
				pFbZAxisRef^.stStatus.bIsMoving := FALSE;
				pFbZAxisRef^.stStatus.bIsHoming := FALSE;
				nErrorID := F_MultiZError_TO_ErrorId(pFbZAxisRef^.stInput.nError);
				bBusy := FALSE;
				bError := TRUE;
				nState := 99;	//go in errorstate
				RETURN;
			ELSE
				pFbZAxisRef^.stStatus.bIsHomed := pFbZAxisRef^.stInput.nStatus.6;
				pFbZAxisRef^.stStatus.bIsHoming := FALSE;
				bBusy := FALSE;
				nState := 9;
			END_IF
	END_CASE
ELSE
	bMoveToHome := FALSE;
	bError := FALSE;
	nErrorId := 0;
	nState := 0;
	timeOut(IN:= FALSE);
	IF pFbZAxisRef > 0 THEN
		pFbZAxisRef^.stStatus.bIsHoming := FALSE;
		pFbZAxisRef^.stOutput.nCtrl := 0;	//Fahrauftrag zurücksetzen (notwendig bei Cancel)	
		IF pFbZAxisRef^.stOutput.nMode = 6 THEN
			pFbZAxisRef^.stOutput.nMode := 0;
		END_IF
	END_IF
	bBusy := FALSE;
END_IF

END_FUNCTION_BLOCK

// ---- Hardware/MultiZ/FB_ZM_Move.TcPOU
FUNCTION_BLOCK FB_ZM_Move
VAR_INPUT
	bExecute		: BOOL;
	rPosition		: REAL;	//Zielposition bzw. Distance bei relativer Fahrt
	rSpeed			: REAL;	//Geschwindigkeit
	eMoveMode		: E_MoveMode;
	pfbZAxisRef		: POINTER TO FB_ZAxisRef;
END_VAR

VAR_OUTPUT
	bBusy			: BOOL;
	bCommandAborted	: BOOL;
	bError			: BOOL;
	nErrorID		: ERRORID;
END_VAR

VAR
	nState				: USINT;
	rCurrentPosition	: REAL;
	tWaitForTrgtReached	: TIME;
	timeOut				: TON;
	fbSdoRead			: FB_SDO_READ;
END_VAR

IF bExecute THEN
	IF pfbZAxisRef = 0 THEN
		nErrorId := E_ErrorIdMultiZ.ERRORID_InvalidZChannel;
		bBusy := FALSE;
		bError := TRUE;
		nState := 99;
		RETURN;
	END_IF
	
	//Wird Achse momentan von anderem Movebaustein genutzt?
	IF (pfbZAxisRef^.pCurrentFb > 0) AND (pfbZAxisRef^.pCurrentFb <> THIS) THEN //wird von anderem FB genutzt
		RETURN;
	END_IF
	
	IF pFbZAxisRef^.stInput.nStatus.3 THEN //Error
		pFbZAxisRef^.stStatus.bError := TRUE;
		pFbZAxisRef^.stOutput.nMode := 0;
		pFbZAxisRef^.stOutput.nCtrl := 0;
		timeOut(IN:= FALSE);
		nErrorID := F_MultiZError_TO_ErrorId(pFbZAxisRef^.stInput.nError);
		bBusy := FALSE;
		bError := TRUE;
		nState := 99;
		RETURN;
	END_IF
	
	IF pFbZAxisRef^.stStatus.bError THEN
		nErrorID := F_MultiZError_TO_ErrorId(pFbZAxisRef^.stInput.nError);
		bBusy := FALSE;
		bError := TRUE;
		nState := 99;
		RETURN;
	END_IF

	//Wenn durch anderen FB Achse gestoppt, dann abbrechen
	IF pFbZAxisRef^.stStatus.bCmdAborted THEN	//Muss noch irgendwo gesetzt werden!!!!
		bCommandAborted := TRUE;
		bBusy := FALSE;
	END_IF
	
	IF timeOut.Q THEN
		timeOut(IN:= FALSE);
		bError := TRUE;
		bBusy := FALSE;
		pFbZAxisRef^.stStatus.bError := TRUE;
		pFbZAxisRef^.stOutput.nCtrl.1 := TRUE;	//Stopbit setzen
		
		CASE nState OF
			2: //Timeout wait for setpointacknowledge
				nErrorId := E_ErrorIdMultiZ.ERRORID_ToWaitSetPointAck;
			3: //Timeout wait for targetreached
				nErrorId := E_ErrorIdMultiZ.ERRORID_ToWaitTrgtReached;
		ELSE
			nErrorId := E_ErrorIdMultiZ.ERRORID_UnknownError;	
		END_CASE
		nState := 99;
		RETURN;
	END_IF		
	
	CASE nState OF
		0:	bBusy := TRUE;
			//Wenn Achse schon aktiv, warten bis wieder frei
			(*IF pstMultiZRef^.stZAxisStatus[nChannel].bHasJob THEN
				RETURN;
			END_IF*)
			pfbZAxisRef^.pCurrentFb := THIS; 
		
			//Geschwindigkeit innerhalb zulässiger Grenzen?
			IF rSpeed <= 0.0 OR rSpeed > pFbZAxisRef^.P_rMaxSpeed THEN
				nErrorID := E_ErrorIdCmd.ERRORID_VelocityOutOfRange;
				bBusy := FALSE;
				bError := TRUE;
				nState := 99;
				RETURN;
			END_IF
			
			pFbZAxisRef^.stStatus.bIsMoving := TRUE;
			pFbZAxisRef^.stStatus.bHasJob := TRUE;
			
			//Aktuelle Position holen
			rCurrentPosition := pFbZAxisRef^.P_rCurrentPos;

			//Targetposition innerhalb zulässiger Grenzen?
			CASE eMoveMode OF
				E_MoveMode.MODE_Relative,E_MoveMode.MODE_Measure:
					IF (rCurrentPosition + rPosition) < pFbZAxisRef^.P_rMinPos OR (rCurrentPosition + rPosition) > pFbZAxisRef^.P_rMaxPos THEN
						nErrorID := E_ErrorIdCmd.ERRORID_TargetPosOutOfRangeZ;
						bError := TRUE;
						bBusy := FALSE;
						nState := 99;
					ELSE
						//Timeout-Zeit für Wait for Targetreached berechnen
						IF eMoveMode = E_MoveMode.MODE_Measure THEN
							//Measure hat fixe Speed "15000"
							tWaitForTrgtReached := REAL_TO_TIME(ABS(rPosition) / 15000 * 1000 + 2000);
						ELSE
							tWaitForTrgtReached := REAL_TO_TIME(ABS(rPosition) / rSpeed * 1000.0 + 2000.0);
						END_IF
					END_IF				

				E_MoveMode.MODE_AbsWithOffset,E_MoveMode.MODE_AbsNoneOffset,E_MoveMode.MODE_Free,E_MoveMode.MODE_Home:
					IF eMoveMode = E_MoveMode.MODE_Home THEN
						rPosition := pFbZAxisRef^.P_rHomePos;
					END_IF
					
					IF rPosition < pFbZAxisRef^.P_rMinPos OR rPosition > pFbZAxisRef^.P_rMaxPos THEN
						nErrorID := E_ErrorIdCmd.ERRORID_TargetPosOutOfRangeZ;
						bError := TRUE;
						bBusy := FALSE;
						nState := 99;
					ELSE
						//Timeout-Zeit für Wait for Targetreached berechnen
						tWaitForTrgtReached := REAL_TO_TIME(ABS(rCurrentPosition - rPosition) / rSpeed * 1000.0 + 2000.0);
					END_IF				
			END_CASE
			
			IF NOT bError THEN
				//Betriebsart Positionsmodus und TargetPos setzen
				IF eMoveMode = E_MoveMode.MODE_Measure THEN
					pFbZAxisRef^.stOutput.nMode := 5;  //Measure
					//Zielposition setzen
					pFbZAxisRef^.P_rRelTargetPos := rPosition;
				ELSIF eMoveMode = E_MoveMode.MODE_Relative THEN
					pFbZAxisRef^.stOutput.nMode := 1;  //Positioniermodus
					//Zielposition setzen
					pFbZAxisRef^.P_rRelTargetPos := rPosition;
				ELSE
					pFbZAxisRef^.stOutput.nMode := 1;
					//Zielposition setzen
					pFbZAxisRef^.P_rAbsTargetPos := rPosition;
				END_IF
				//Geschwindigkeit setzen
				pFbZAxisRef^.stOutput.nVelo := REAL_TO_DINT(rSpeed);
				nState := 1;
			END_IF

		1:	//Fahrauftrag starten
			IF eMoveMode = E_MoveMode.MODE_Relative THEN	//Relativ
				pFbZAxisRef^.stOutput.nCtrl := 5;
			ELSE
				pFbZAxisRef^.stOutput.nCtrl := 1;	
			END_IF
			nState := 2;
	
		2:	//SetpointAcknowledge?
			IF pFbZAxisRef^.stInput.nStatus.1 THEN
				pFbZAxisRef^.stOutput.nCtrl.0 := FALSE;	//Fahrauftrag zurücksetzen
				timeOut(IN:= FALSE);
				nState := 3;
			ELSE
				timeOut(IN:= TRUE, PT:=T#1200MS);	//Timer für Timeout starten
			END_IF
			
		3:	//TargetReached?
			//IF pFbZAxisRef^.stInput.nStatus.0 THEN
			IF pFbZAxisRef^.stInput.nStatus = 193 THEN
				timeOut(IN:= FALSE);
				IF eMoveMode = E_MoveMode.MODE_Measure THEN
					nState := 4;
				ELSE
					bBusy := FALSE;	
				END_IF
			ELSE
				timeOut(IN:= TRUE, PT:= tWaitForTrgtReached);	//Timer für Timeout starten
			END_IF
		
		4:	//wenn "MODE_Measure", dann ZOffset holen
			fbSdoRead(sADSNetID:= pFbZAxisRef^.pMultiZRef^.P_sAdsNetId,	nPortNr:= pFbZAxisRef^.pMultiZRef^.P_nAdsPort,
					nIndex:= cZSensOffset.nIndex, nSubIndex:= pFbZAxisRef^.nChannel, nDataLength:= cZSensOffset.nLength, bExecute:= TRUE);
			IF NOT fbSdoRead.bBusy THEN
				IF fbSdoRead.bError THEN
					bError := TRUE;
					nState := 99;
				ELSE
					pFbZAxisRef^.P_nZSensorID := fbSdoRead.nData;
				END_IF
				fbSdoRead(bExecute:= FALSE);
				bBusy := FALSE;
			END_IF
	END_CASE
ELSE
	bBusy := FALSE;
	nState := 0;
	bError := FALSE;
	nErrorID := 0;
	timeOut(IN:= FALSE);
	IF pfbZAxisRef^.pCurrentFb > 0 THEN
		IF pfbZAxisRef^.pCurrentFb = THIS THEN
			pfbZAxisRef^.pCurrentFb := 0;
			pFbZAxisRef^.stStatus.bCmdAborted := FALSE;
			pFbZAxisRef^.stOutput.nMode := 0;
			pFbZAxisRef^.stStatus.bHasJob := FALSE;
			pFbZAxisRef^.stStatus.bIsMoving := FALSE;		
		END_IF		
	END_IF
END_IF

END_FUNCTION_BLOCK

// ---- Hardware/MultiZ/FB_ZM_Stop.TcPOU
FUNCTION_BLOCK FB_ZM_Stop
VAR_INPUT
	bExecute		: BOOL;
	pFbZAxisRef		: POINTER TO FB_ZAxisRef;
END_VAR

VAR_OUTPUT
	bBusy			: BOOL;
	bError			: BOOL;
	nErrorID		: ERRORID;
END_VAR

VAR
	nState				: USINT;
	timeOut				: TON;
	nCurrentPosition	: REAL;
	//bFlagGetPosition 	: BOOL := TRUE;
	//fbMultiZReadSdoVar	: FB_MultiZReadSdoVar;
END_VAR

IF bExecute THEN
	IF pFbZAxisRef = 0 THEN
		nErrorId := E_ErrorIdMultiZ.ERRORID_InvalidZChannel;
		bError := TRUE;
		nState := 99;	//go in errorstate		
		RETURN;
	END_IF
	
	IF pFbZAxisRef^.stInput.nStatus.3 THEN //Error
		pFbZAxisRef^.stStatus.bError := TRUE;
		pFbZAxisRef^.stOutput.nMode := 0;
		pFbZAxisRef^.stOutput.nCtrl := 0;
		timeOut(IN:= FALSE);
		nErrorID := F_MultiZError_TO_ErrorId(pFbZAxisRef^.stInput.nError);
		bBusy := FALSE;
		bError := TRUE;
		nState := 99;	//go in errorstate
		RETURN;
	END_IF

	IF timeOut.Q THEN
		timeOut(IN:= FALSE);
		bError := TRUE;
		bBusy := FALSE;
		pFbZAxisRef^.stStatus.bError := TRUE;
		pFbZAxisRef^.stOutput.nMode := 0;
		pFbZAxisRef^.stOutput.nCtrl := 0;
		nErrorId := E_ErrorIdMultiZ.ERRORID_ToWaitStop;
		nState := 99;	//go in errorstate
		RETURN;
	END_IF		

	CASE nState OF		
		0:	bBusy := TRUE;	
			pFbZAxisRef^.stStatus.bCmdAborted := TRUE;
			//Stoppen	
			pFbZAxisRef^.stOutput.nCtrl.1 := TRUE;	//Stopbit setzen
			nState := 1;
			
		1:	//Stopbit gesetzt?
			IF pFbZAxisRef^.stInput.nStatus.2 THEN
				timeOut(IN:= FALSE);
				pFbZAxisRef^.stOutput.nMode := 0;
				pFbZAxisRef^.stOutput.nCtrl.1 := FALSE;	//Stopbit zurücksetzen
				pFbZAxisRef^.stOutput.nCtrl.0 := FALSE;	//Fahrauftrag zurücksetzen
				nState := 80;
				bBusy := FALSE;
			ELSE
				timeOut(IN:= TRUE, PT:=T#1000MS);	//Timer für Timeout starten
			END_IF
	END_CASE
ELSE
	nState := 0;
	bBusy := FALSE;
	timeOut(IN:= FALSE);
	bError := FALSE;
	nErrorID := 0;
END_IF

END_FUNCTION_BLOCK

// ---- Objects/Targets/Passive/FB_Mtp.TcPOU
{attribute 'enable_dynamic_creation'}
FUNCTION_BLOCK FB_Mtp EXTENDS FB_Array
VAR_INPUT
END_VAR
VAR_OUTPUT
END_VAR
VAR
	rOffsetCol1		: REAL;			//Abstand Spalte 1 vom linken MTP-Rand (Mitte Well)
	rOffsetRow1		: REAL;			//Abstand Zeile 1 vom oberen MTP-Rand (Mitte Well)
	rSpaceCols		: REAL;			//Abstand Spalten zueinander (Mitte Wells)
	rSpaceRows		: REAL;			//Abstand Zeilen zueinander (Mitte Wells)	
	rWellDiameter	: REAL;			//Welldurchmesser
	rWellDepth		: REAL;			//Welltiefe
	stOffsetWell1	: ST_3DPoint;	//Korrekturoffset linkes unteres Well
	rFactorCols		: REAL := 1;	//Faktor auf Abstand von erster Spalte zu letzer Spalte (durch teachen oder manuell)
	rFactorRows		: REAL := 1;	//Faktor auf Abstand von unterster Zeile zu oberster Zeile (durch teachen oder manuell)
	nGCodeTargetNr	: UINT;
END_VAR

METHOD FB_init : BOOL
VAR_INPUT
	bInitRetains : BOOL; // if TRUE, the retain variables are initialized (warm start / cold start)
	bInCopyCode : BOOL;  // if TRUE, the instance afterwards gets moved into the copy code (online change)
END_VAR
eObjectType := E_ObjectType.OBJECTTYPE_Mtp;
eObjectGroup := E_ObjectGroup.OBJECTGROUP_Target OR E_ObjectGroup.OBJECTGROUP_Array;
END_METHOD

METHOD M_AddChild : ERRORID
VAR_INPUT
	pObject : POINTER TO FB_Object;
	nSlotNr	: UINT;
	nIndex 	: INT;
END_VAR
//Kann folgende Objekte aufnehmen:
//Points
IF pObject > 0 THEN
	IF pObject^.P_eObjectType = E_ObjectType.OBJECTTYPE_Point OR pObject^.P_eObjectType = E_ObjectType.OBJECTTYPE_Slide THEN
		M_AddChild := SUPER^.M_AddChild(pObject,nSlotNr,nIndex);
	ELSE
		M_AddChild := E_ErrorIdObjMgmt.ERRORID_InvalidParentObject;
	END_IF
ELSE
	M_AddChild := E_ErrorIdObjMgmt.ERRORID_InvalidParentObject;
END_IF
END_METHOD

METHOD M_CalcKorrFactor : ERRORID
VAR_INPUT
	stAbsPos : ST_3DPoint;
END_VAR

VAR
	stTempPoint : ST_3DPoint;
	rTheoDistance : REAL;
	rRealDistance : REAL;
END_VAR
{warning 'siehe Kommentar'}
//hier muss auch noch auf eine spätere Verdrehung geachtet werden
stTempPoint := P_stAbsPosLB;
rTheoDistance := (nCols - 1) * rSpaceCols;
rRealDistance := stAbsPos.X - (stTempPoint.X + rOffsetCol1 + stOffsetWell1.X);
rFactorCols := rRealDistance / rTheoDistance;
rTheoDistance := (nRows - 1) * rSpaceRows;
rRealDistance := stAbsPos.Y - (stTempPoint.Y + rOffsetRow1 + stOffsetWell1.Y);
rFactorRows := rRealDistance / rTheoDistance;
(*
von wo wird diese Methode aufgerufen?
-> in TeachTarget nachdem das rechte obere Well eingeteached wurde
-> man muss aber davon ausgehen, dass die MTP verdreht ist oder zumindest auf einem verdrehtem Parent sitzt
-> als erstes wäre jetzt mal interessant zu wissen, ob das für eine Mtp überhaupt ein Thema ist?
-> definitiv sollte ein TargetTray verdrehbar sein, da in der Linie 


*)
END_METHOD

METHOD M_CalcOffsetWellLB : ERRORID
VAR_INPUT
	stAbsPos : ST_3DPoint;
	nZLevel	 : USINT; 
END_VAR

VAR
	stTempPoint : ST_3DPoint;
END_VAR
stTempPoint := P_stAbsPosLB;
stTempPoint.X := stTempPoint.X + rOffsetCol1;
stTempPoint.Y := stTempPoint.Y + rOffsetRow1;
stOffsetWell1.X := stAbsPos.X - stTempPoint.X;
stOffsetWell1.Y := stAbsPos.Y - stTempPoint.Y;
IF nZLevel = 0 THEN	//PrePos
	stOffsetWell1.Z := stAbsPos.Z - stTempPoint.Z;
ELSIF nZLevel = 1 THEN //WorkPos
	//stTempPoint := M_GetAbsPoint(eTargetRef:= E_TargetRef.TARGETREF_TwoDimArray, nParam1:= 1, nParam2:= 1, nParam3:= 0, nZLevel:= 0, nErrorId=> nErrorId);
	//hier stellt sich die Frage, wie der Offset angegeben wird falls das Parent verdreht ist
	//vorerst wird das nicht beachtet, da momentan nur Slides gedreht werden
	stTempPoint := M_GetAbsPos(pchildPos:= 0 ,eTargetRef:= E_TargetRef.TARGETREF_TwoDimArray, nParam1:= 1, nParam2:= 1, nParam3:= 0, nParam4:= 0, nZLevel:= 0(*, nErrorId=> nErrorId*));
	rWellDepth :=  stTempPoint.Z - stAbsPos.Z;
END_IF
END_METHOD

METHOD M_CheckAction : ERRORID
VAR_INPUT
	refActionData 	: REFERENCE TO ST_ActionData;
	pCorrelObject	: POINTER TO FB_Object;
END_VAR
IF refActionData.eAction = E_Action.ACTION_TeachTarget THEN
	IF DINT_TO_UINT(refActionData.aParams[1]) <> E_TargetRef.TARGETREF_TwoDimArray THEN
		M_CheckAction := E_ErrorIdCmd.ERRORID_InvalidTargetPointRef;
	END_IF
END_IF
END_METHOD

METHOD M_GetAbsPos : ST_3DPoint
VAR_INPUT
	pChildPos	: POINTER TO ST_3DPoint;
	eTargetRef 	: E_TargetRef;
	nParam1		: UINT;
 	nParam2		: UINT;
	nParam3		: USINT;
	nParam4		: USINT;
	nZLevel		: USINT;
END_VAR
VAR_OUTPUT
	nErrorId 	: ERRORID;
	lrAngle		: LREAL;
END_VAR
VAR
	stLocPosLB : ST_3DPoint;
	nCol : UINT;
	nRow : UINT;	
END_VAR
IF eTargetRef = E_TargetRef.TARGETREF_TwoDimArray THEN
	//Checken ob gültige Spalte und Zeile
	IF nParam1 = 0 OR nParam1 > nCols THEN
		nErrorId := E_ErrorIdCmd.ERRORID_InvalidTargetPointCol;
		RETURN;
	END_IF
	IF nParam2 = 0 OR nParam2 > nRows THEN
		nErrorId := E_ErrorIdCmd.ERRORID_InvalidTargetPointRow;
		RETURN;
	END_IF
	
	stLocPosLB := P_stRelPosLB;	//hier wird auch berücksichtigt, wenn die Mtp an einem Slot hängt
	//relative X-Position berechnen
	stLocPosLB.X := stLocPosLB.X + rOffsetCol1 + (rSpaceCols * (nParam1 - 1) * rFactorCols);
	//relative Y-Position berechnen
	stLocPosLB.Y := stLocPosLB.Y + rOffsetRow1 + (rSpaceRows * (nRows - nParam2) * rFactorRows);
	//Offset vom Well1 dazurechnen
	stLocPosLB := F_Add3DPoints(stLocPosLB,stOffsetWell1);
	IF nZLevel = 1 THEN  //WorkPos
		stLocPosLB.Z := stLocPosLB.Z - rWellDepth;
	END_IF
	
	M_GetAbsPos := pParentTarget^.M_GetAbsPos(pChildPos := ADR(stLocPosLB), eTargetRef:= E_TargetRef.TARGETREF_LeftBottom,
													nParam1:= 0,
													nParam2:= 0, nParam3:= 0, nParam4:= 0, nZLevel:= 0,
													lrAngle => lrAngle, nErrorId=> nErrorId);
													
ELSIF eTargetRef = E_TargetRef.TARGETREF_SequParaToArrayItem THEN
	//das Item muss 0 und <= Zeilen*Spalten sein
	IF nParam1 > 0 AND nParam1 <= nCols * nRows THEN
		nRow := nParam1 MOD nCols;
		IF nRow > 0 THEN
			nRow := (nParam1 - nRow) / nCols + 1;
		ELSE
			nRow := (nParam1 - nRow) / nCols;
		END_IF
		nCol := nParam1 - nCols * (nRow - 1);
		
		stLocPosLB := P_stRelPosLB;	//hier wird auch berücksichtigt, wenn die Mtp an einem Slot hängt
		//relative X-Position berechnen
		stLocPosLB.X := stLocPosLB.X + rOffsetCol1 + (rSpaceCols * (nCol - 1) * rFactorCols);
		//relative Y-Position berechnen
		stLocPosLB.Y := stLocPosLB.Y + rOffsetRow1 + (rSpaceRows * (nRows - nRow) * rFactorRows);
		//Offset vom Well1 dazurechnen
		stLocPosLB := F_Add3DPoints(stLocPosLB,stOffsetWell1);
		IF nZLevel = 1 THEN  //WorkPos
			stLocPosLB.Z := stLocPosLB.Z - rWellDepth;
		END_IF
		
		M_GetAbsPos := pParentTarget^.M_GetAbsPos(pChildPos := ADR(stLocPosLB), eTargetRef:= E_TargetRef.TARGETREF_LeftBottom,
														nParam1:= 0,
														nParam2:= 0, nParam3:= 0, nParam4:= 0, nZLevel:= 0,
														lrAngle => lrAngle, nErrorId=> nErrorId);		
	ELSE
		nErrorId := E_ErrorIdCmd.ERRORID_InvalidArrayItem;
	END_IF
ELSE
	M_GetAbsPos := SUPER^.M_GetAbsPos(pChildPos := pChildPos, eTargetRef:= eTargetRef,
													nParam1:= nParam1,
													nParam2:= nParam2, nParam3:= nParam3, nParam4:= 0, nZLevel:= nZLevel,
													lrAngle => lrAngle, nErrorId=> nErrorId);		
END_IF
END_METHOD

METHOD M_GetAllProps : ERRORID
VAR_INPUT
	refCmdData : REFERENCE TO  ST_CmdData;
END_VAR
SUPER^.M_GetAllProps(refCmdData);

nCurrentPropIndex := nCurrentPropIndex + 1;
refCmdData.n32Data[nCurrentPropIndex] := REAL_TO_DINT(rOffsetCol1);
nCurrentPropIndex := nCurrentPropIndex + 1;
refCmdData.n32Data[nCurrentPropIndex] := REAL_TO_DINT(rOffsetRow1);
nCurrentPropIndex := nCurrentPropIndex + 1;
refCmdData.n32Data[nCurrentPropIndex] := REAL_TO_DINT(rSpaceCols);
nCurrentPropIndex := nCurrentPropIndex + 1;
refCmdData.n32Data[nCurrentPropIndex] := REAL_TO_DINT(rSpaceRows);
nCurrentPropIndex := nCurrentPropIndex + 1;
refCmdData.n32Data[nCurrentPropIndex] := REAL_TO_DINT(rWellDiameter);
nCurrentPropIndex := nCurrentPropIndex + 1;
refCmdData.n32Data[nCurrentPropIndex] := REAL_TO_DINT(rWellDepth);
nCurrentPropIndex := nCurrentPropIndex + 1;
refCmdData.n32Data[nCurrentPropIndex] := REAL_TO_DINT(stOffsetWell1.X);
nCurrentPropIndex := nCurrentPropIndex + 1;
refCmdData.n32Data[nCurrentPropIndex] := REAL_TO_DINT(stOffsetWell1.Y);
nCurrentPropIndex := nCurrentPropIndex + 1;
refCmdData.n32Data[nCurrentPropIndex] := REAL_TO_DINT(stOffsetWell1.Z);
nCurrentPropIndex := nCurrentPropIndex + 1;
refCmdData.n32Data[nCurrentPropIndex] := REAL_TO_DINT(rFactorCols * 1000000.0);
nCurrentPropIndex := nCurrentPropIndex + 1;
refCmdData.n32Data[nCurrentPropIndex] := REAL_TO_DINT(rFactorRows * 1000000.0);
nCurrentPropIndex := nCurrentPropIndex + 1;
refCmdData.n32Data[nCurrentPropIndex] := nGCodeTargetNr;
END_METHOD

METHOD M_GetRectIsInnerWell : BOOL
VAR_INPUT
	stRectArea : FB_Rectangle;
END_VAR

VAR
	nCol : UINT;
	nRow : UINT;
	stCircle : ST_Circle;
	stPoint : ST_3DPoint;
END_VAR
stCircle.rD := rWellDiameter;

//Alle Wells durchlaufen
FOR nCol := 1 TO nCols BY 1 DO
	FOR nRow := 1 TO nRows BY 1 DO
		stPoint := M_GetAbsPos(0,E_TargetRef.TARGETREF_TwoDimArray,nCol,nRow,0,0,0);
		stCircle.rX := stPoint.X;
		stCircle.rY := stPoint.Y;
		IF F_RectInnerCircle(stRectArea,stCircle) THEN
			M_GetRectIsInnerWell := TRUE;
			RETURN;
		END_IF
	END_FOR
END_FOR
END_METHOD

METHOD M_SetAllProps : ERRORID
VAR_INPUT
	refCmdData : REFERENCE TO  ST_CmdData;
END_VAR
M_SetAllProps := SUPER^.M_SetAllProps(refCmdData);

IF M_SetAllProps > 0 THEN
	RETURN;
END_IF

nCurrentPropIndex := nCurrentPropIndex + 1;
nSpecPropIndex := nCurrentPropIndex; 
rOffsetCol1 := DINT_TO_REAL(refCmdData.n32Data[nCurrentPropIndex]);
nCurrentPropIndex := nCurrentPropIndex + 1;
rOffsetRow1 := DINT_TO_REAL(refCmdData.n32Data[nCurrentPropIndex]);
nCurrentPropIndex := nCurrentPropIndex + 1;
rSpaceCols := DINT_TO_REAL(refCmdData.n32Data[nCurrentPropIndex]);
nCurrentPropIndex := nCurrentPropIndex + 1;
rSpaceRows := DINT_TO_REAL(refCmdData.n32Data[nCurrentPropIndex]);
nCurrentPropIndex := nCurrentPropIndex + 1;
rWellDiameter := DINT_TO_REAL(refCmdData.n32Data[nCurrentPropIndex]);
nCurrentPropIndex := nCurrentPropIndex + 1;
rWellDepth := DINT_TO_REAL(refCmdData.n32Data[nCurrentPropIndex]);
nCurrentPropIndex := nCurrentPropIndex + 1;
stOffsetWell1.X := DINT_TO_REAL(refCmdData.n32Data[nCurrentPropIndex]);
nCurrentPropIndex := nCurrentPropIndex + 1;
stOffsetWell1.Y := DINT_TO_REAL(refCmdData.n32Data[nCurrentPropIndex]);
nCurrentPropIndex := nCurrentPropIndex + 1;
stOffsetWell1.Z := DINT_TO_REAL(refCmdData.n32Data[nCurrentPropIndex]);
nCurrentPropIndex := nCurrentPropIndex + 1;
rFactorCols := DINT_TO_REAL(refCmdData.n32Data[nCurrentPropIndex]) / 1000000.0;
nCurrentPropIndex := nCurrentPropIndex + 1;
rFactorRows := DINT_TO_REAL(refCmdData.n32Data[nCurrentPropIndex]) / 1000000.0;
nCurrentPropIndex := nCurrentPropIndex + 1;
nGCodeTargetNr := DINT_TO_UINT(refCmdData.n32Data[nCurrentPropIndex]);
nNoOfProps := nCurrentPropIndex + 1;
END_METHOD

METHOD M_SetSingleProp : ERRORID
VAR_INPUT
	refCmdData : REFERENCE TO  ST_CmdData;
END_VAR
IF nSpecPropIndex = refCmdData.aHeader[1] THEN
	rOffsetCol1 := DINT_TO_REAL(refCmdData.n32Data[0]);
ELSIF (nSpecPropIndex + 1) = refCmdData.aHeader[1] THEN
	rOffsetRow1 := DINT_TO_REAL(refCmdData.n32Data[0]);
ELSIF (nSpecPropIndex + 2) = refCmdData.aHeader[1] THEN
	rSpaceCols := DINT_TO_REAL(refCmdData.n32Data[0]);
ELSIF (nSpecPropIndex + 3) = refCmdData.aHeader[1] THEN
	rSpaceRows := DINT_TO_REAL(refCmdData.n32Data[0]);
ELSIF (nSpecPropIndex + 4) = refCmdData.aHeader[1] THEN
	rWellDiameter := DINT_TO_REAL(refCmdData.n32Data[0]);
ELSIF (nSpecPropIndex + 5) = refCmdData.aHeader[1] THEN
	rWellDepth := DINT_TO_REAL(refCmdData.n32Data[0]);
ELSIF (nSpecPropIndex + 6) = refCmdData.aHeader[1] THEN
	stOffsetWell1.X := DINT_TO_REAL(refCmdData.n32Data[0]);
ELSIF (nSpecPropIndex + 7) = refCmdData.aHeader[1] THEN
	stOffsetWell1.Y := DINT_TO_REAL(refCmdData.n32Data[0]);
ELSIF (nSpecPropIndex + 8) = refCmdData.aHeader[1] THEN
	stOffsetWell1.Z := DINT_TO_REAL(refCmdData.n32Data[0]);
ELSIF (nSpecPropIndex + 9) = refCmdData.aHeader[1] THEN
	rFactorCols := DINT_TO_REAL(refCmdData.n32Data[0]) / 1000000.0;
ELSIF (nSpecPropIndex + 10) = refCmdData.aHeader[1] THEN
	rFactorRows := DINT_TO_REAL(refCmdData.n32Data[0]) / 1000000.0;
ELSE
	M_SetSingleProp := SUPER^.M_SetSingleProp(refCmdData);
END_IF
END_METHOD

PROPERTY P_nCols : UINT
GET
P_nCols := nCols;
END_GET
END_PROPERTY

PROPERTY P_nGCodeTargetNr : UINT
GET
P_nGCodeTargetNr := nGCodeTargetNr;
END_GET
END_PROPERTY

PROPERTY P_nRows : UINT
GET
P_nRows := nRows;
END_GET
END_PROPERTY

PROPERTY P_rSpaceRows : REAL
GET
P_rSpaceRows := rSpaceRows;
END_GET
END_PROPERTY

END_FUNCTION_BLOCK

// ---- Objects/Targets/Passive/FB_Array.TcPOU
FUNCTION_BLOCK FB_Array EXTENDS FB_TargetBase
VAR_INPUT
END_VAR
VAR_OUTPUT
END_VAR
VAR
	nCols			: UINT;		//Anzahl Spalten
	nRows			: UINT;		//Anzahl Zeilen
	nPropIndexCols  : UINT;
END_VAR

METHOD M_CheckAction : ERRORID
VAR_INPUT
	refActionData : REFERENCE TO ST_ActionData;
	pCorrelObject	: POINTER TO FB_Object;
END_VAR
IF refActionData.eAction = E_Action.ACTION_TeachTarget THEN
	IF DINT_TO_UINT(refActionData.aParams[1]) <> E_TargetRef.TARGETREF_TwoDimArray THEN
		M_CheckAction := E_ErrorIdCmd.ERRORID_InvalidTargetPointRef;
	END_IF
END_IF
END_METHOD

METHOD M_GetAbsPos : ST_3DPoint
VAR_INPUT
	pChildPos	: POINTER TO ST_3DPoint;
	eTargetRef 	: E_TargetRef;
	nParam1		: UINT;
 	nParam2		: UINT;
	nParam3		: USINT;
	nParam4		: USINT;
	nZLevel		: USINT;
END_VAR
VAR_OUTPUT
	nErrorId 	: ERRORID;
	lrAngle		: LREAL;
END_VAR
VAR
	stLocPos : ST_3DPoint;
	rTemp : REAL;
	nCol : UINT;
	nRow : UINT;
END_VAR
IF eTargetRef = E_TargetRef.TARGETREF_TwoDimArray THEN
	//Checken ob gültige Spalte und Zeile
	IF nParam1 = 0 OR nParam1 > nCols THEN
		nErrorId := E_ErrorIdCmd.ERRORID_InvalidTargetPointCol;
		RETURN;
	END_IF
	IF nParam2 = 0 OR nParam2 > nRows THEN
		nErrorId := E_ErrorIdCmd.ERRORID_InvalidTargetPointRow;
		RETURN;
	END_IF
	
	stLocPos := stRelPos;
	//relative X-Position berechnen
	IF ncols > 1 THEN
		rTemp := stDimension.Width / (nCols - 1); //Spaltenbreite	
	END_IF
	stLocPos.X := stLocPos.X + rTemp * nParam1 - rTemp;
	
	//relative Y-Position berechnen
	IF nRows > 1 THEN
		rTemp := stDimension.Depth / (nRows - 1); //Zeilenhöhe
		stLocPos.Y := stLocPos.Y + stDimension.Depth - rTemp * nParam2 + rTemp;
	END_IF
	
	
	
	M_GetAbsPos := pParentTarget^.M_GetAbsPos(pChildPos := ADR(stLocPos), eTargetRef:= E_TargetRef.TARGETREF_LeftBottom,
													nParam1:= 0,
													nParam2:= 0, nParam3:= 0, nParam4:= 0, nZLevel:= 0,
													lrAngle => lrAngle, nErrorId=> nErrorId);
													
ELSIF eTargetRef = E_TargetRef.TARGETREF_SequParaToArrayItem THEN
	//das Item muss 0 und <= Zeilen*Spalten sein
	IF nParam1 > 0 AND nParam1 <= nCols * nRows THEN
		nRow := nParam1 MOD nCols; 
		IF nRow > 0 THEN
			nRow := (nParam1 - nRow) / nCols + 1;
		ELSE
			nRow := (nParam1 - nRow) / nCols;
		END_IF
		nCol := nParam1 - nCols * (nRow - 1);
		
		stLocPos := stRelPos;
		//relative X-Position berechnen
		IF ncols > 1 THEN
			rTemp := stDimension.Width / (nCols - 1); //Spaltenbreite	
		END_IF
		stLocPos.X := stLocPos.X + rTemp * nCol - rTemp;
		
		//relative Y-Position berechnen
		IF nRows > 1 THEN
			rTemp := stDimension.Depth / (nRows - 1); //Zeilenhöhe
			stLocPos.Y := stLocPos.Y + stDimension.Depth - rTemp * nRow + rTemp;
		END_IF
		
		
		
		M_GetAbsPos := pParentTarget^.M_GetAbsPos(pChildPos := ADR(stLocPos), eTargetRef:= E_TargetRef.TARGETREF_LeftBottom,
														nParam1:= 0,
														nParam2:= 0, nParam3:= 0, nParam4:= 0, nZLevel:= 0,
														lrAngle => lrAngle, nErrorId=> nErrorId);		
	ELSE
		nErrorId := E_ErrorIdCmd.ERRORID_InvalidArrayItem;
	END_IF
ELSE
	M_GetAbsPos := SUPER^.M_GetAbsPos(pChildPos := pChildPos, eTargetRef:= eTargetRef,
													nParam1:= nParam1,
													nParam2:= nParam2, nParam3:= nParam3, nParam4:= 0, nZLevel:= nZLevel,
													lrAngle => lrAngle, nErrorId=> nErrorId);	
END_IF
END_METHOD

METHOD M_GetAllProps : ERRORID
VAR_INPUT
	refCmdData : REFERENCE TO  ST_CmdData;
END_VAR
SUPER^.M_GetAllProps(refCmdData);
nCurrentPropIndex := nCurrentPropIndex + 1;
refCmdData.n32Data[nCurrentPropIndex] := nCols;
nCurrentPropIndex := nCurrentPropIndex + 1;
refCmdData.n32Data[nCurrentPropIndex] := nRows;
END_METHOD

METHOD M_GetNextArrayIndex : BOOL
VAR_INPUT
	eOrder	  : E_ArrayOrder;
	nStartCol : UINT;
	nStartRow : UINT;
END_VAR
VAR_OUTPUT
	nCol : UINT;
	nRow : UINT;
END_VAR
CASE eOrder OF
	E_ArrayOrder.RowWiseSaw:
		IF nStartCol = 0 THEN //Start
			nCol := 1;
			nRow := 1;
			M_GetNextArrayIndex := TRUE;
		ELSE
			//Zeile darf nicht "0" sein
			IF nStartRow = 0 THEN
				RETURN;
			END_IF
			//Letzte Spalte?
			IF (nStartCol = nCols) THEN //Zeilenvorschub
				nCol := 1;
				nRow := nStartRow + 1;
				//Zeile darf nicht größer als Anzahl Zeilen sein
				IF nRow > nRows THEN
					nRow := 0;
					RETURN;
				END_IF
			ELSE //Spaltenvorschub
				nCol := nStartCol + 1;
				nRow := nStartRow;
			END_IF
			M_GetNextArrayIndex := TRUE;
		END_IF
	E_ArrayOrder.RowWiseMeander:
		IF nStartCol = 0 THEN //Start
			nCol := 1;
			nRow := 1;
			M_GetNextArrayIndex := TRUE;
		ELSE
			//Zeile darf nicht "0" sein
			IF nStartRow = 0 THEN
				RETURN;
			END_IF
			//StartSpalte die erste oder letzte Spalte?
			IF (nStartCol = nCols AND (nStartRow MOD 2) = 1) OR (nStartCol = 1 AND (nStartRow MOD 2) = 0) THEN //Zeilenvorschub
				nRow := nStartRow + 1;
				//Zeile darf nicht größer als Anzahl Zeilen sein
				IF nRow > nRows THEN
					nRow := 0;
					RETURN;
				END_IF
				nCol := nStartCol;
				M_GetNextArrayIndex := TRUE;
			ELSE
				//Spalte vor oder zurück zählen?
				IF (nStartRow MOD 2 = 0) THEN //gerade -> Spalte zurück zählen
					nCol := nStartCol - 1;
				ELSE //ungerade -> Spalte vorwärts zählen
					nCol := nStartCol + 1;
				END_IF
				M_GetNextArrayIndex := TRUE;
				nRow := nStartRow;
			END_IF
		END_IF	
	E_ArrayOrder.ColWiseSaw:
		IF nStartRow = 0 THEN //Start
			nCol := 1;
			nRow := 1;
			M_GetNextArrayIndex := TRUE;
		ELSE
			//Spalte darf nicht "0" sein
			IF nStartCol = 0 THEN
				RETURN;
			END_IF
			//Letzte Spalte?
			IF (nStartRow = nRows) THEN //Spaltenvorschub
				nRow := 1;
				nCol := nStartCol + 1;
				IF nCol > nCols THEN
					nCol:= 0;
					RETURN;
				END_IF
			ELSE //Zeilenvorschub
				nRow := nStartRow + 1;
				nCol := nStartCol;
			END_IF
			M_GetNextArrayIndex := TRUE;
		END_IF	
	E_ArrayOrder.ColWiseMeander:
		IF nStartRow = 0 THEN //Start
			nCol := 1;
			nRow := 1;
			M_GetNextArrayIndex := TRUE;
		ELSE
			//Spalte darf nicht "0" sein
			IF nStartCol = 0 THEN
				RETURN;
			END_IF
			//StartZeile die erste oder letzte Zeile?
			IF (nStartRow = nRows AND (nStartCol MOD 2) = 1) OR (nStartRow = 1 AND (nStartCol MOD 2) = 0) THEN //Spaltenvorschub
				nCol := nStartCol + 1;
				//Spalte darf nicht größer als Anzahl Spalten sein
				IF nCol > nCols THEN
					nCol := 0;
					RETURN;
				END_IF
				nRow := nStartRow;
				M_GetNextArrayIndex := TRUE;
			ELSE
				//Zeile vor oder zurück zählen?
				IF (nStartCol MOD 2 = 0) THEN //gerade -> Spalte zurück zählen
					nRow := nStartRow - 1;
				ELSE //ungerade -> Spalte vorwärts zählen
					nRow := nStartRow + 1;
				END_IF
				M_GetNextArrayIndex := TRUE;
				nCol := nStartCol;
			END_IF
		END_IF
END_CASE
END_METHOD

METHOD M_SetAllProps : ERRORID
VAR_INPUT
	refCmdData : REFERENCE TO  ST_CmdData;
END_VAR
M_SetAllProps := SUPER^.M_SetAllProps(refCmdData);

IF M_SetAllProps > 0 THEN
	RETURN;
END_IF

nCurrentPropIndex := nCurrentPropIndex + 1;
nPropIndexCols := nCurrentPropIndex;
nCols := DINT_TO_UINT(refCmdData.n32Data[nCurrentPropIndex]);
nCurrentPropIndex := nCurrentPropIndex + 1;
nRows := DINT_TO_UINT(refCmdData.n32Data[nCurrentPropIndex]);

nNoOfProps := nCurrentPropIndex + 1;
END_METHOD

METHOD M_SetSingleProp : ERRORID
VAR_INPUT
	refCmdData : REFERENCE TO  ST_CmdData;
END_VAR
IF nPropIndexCols = refCmdData.aHeader[1] THEN
	nCols := DINT_TO_UINT(refCmdData.n32Data[0]);
ELSIF (nPropIndexCols + 1) = refCmdData.aHeader[1] THEN
	nRows := DINT_TO_UINT(refCmdData.n32Data[0]);
ELSE
	M_SetSingleProp := SUPER^.M_SetSingleProp(refCmdData);
END_IF
END_METHOD

PROPERTY P_nCols : UINT
GET
P_nCols := nCols;
END_GET
END_PROPERTY

PROPERTY P_nRows : UINT
GET
P_nRows := nRows;
END_GET
END_PROPERTY

END_FUNCTION_BLOCK

// ---- Objects/F_RectInnerCircle.TcPOU
FUNCTION F_RectInnerCircle : BOOL
VAR_INPUT
	stRect 		: FB_Rectangle;
	stCircle	: ST_Circle;
END_VAR
VAR
	rSquareRad	: REAL;
	stPoint1	: ST_2DPoint;
	stPoint2	: ST_2DPoint;
	stPoint3	: ST_2DPoint;
	stPoint4	: ST_2DPoint;
END_VAR

//Berechnet, ob sich Rechteck innerhalb eines Kreises befindet
rSquareRad := (stCircle.rD / 2.0) * (stCircle.rD / 2.0);	//Quadrat Radius des Kreises
//Alle Eckpunkte des Rechteckes
stPoint1.X := stRect.X1;
stPoint1.Y := stRect.Y1;
stPoint2.X := stRect.X2;
stPoint2.Y := stRect.Y1;
stPoint3.X := stRect.X2;
stPoint3.Y := stRect.Y2;
stPoint4.X := stRect.X1;
stPoint4.Y := stRect.Y2;
//4* Satz des Pythagoras - überprüfen, ob alle Punkte innerhalb des Kreises
F_RectInnerCircle := 
	((stCircle.rX - stPoint1.X) * (stCircle.rX - stPoint1.X) + (stCircle.rY - stPoint1.Y) * (stCircle.rY - stPoint1.Y)) <= rSquareRad AND
	((stCircle.rX - stPoint2.X) * (stCircle.rX - stPoint2.X) + (stCircle.rY - stPoint2.Y) * (stCircle.rY - stPoint2.Y)) <= rSquareRad AND
	((stCircle.rX - stPoint3.X) * (stCircle.rX - stPoint3.X) + (stCircle.rY - stPoint3.Y) * (stCircle.rY - stPoint3.Y)) <= rSquareRad AND
	((stCircle.rX - stPoint4.X) * (stCircle.rX - stPoint4.X) + (stCircle.rY - stPoint4.Y) * (stCircle.rY - stPoint4.Y)) <= rSquareRad;

END_FUNCTION

// ---- Objects/Tools/FB_MzHead.TcPOU
FUNCTION_BLOCK FB_MzHead EXTENDS FB_MzBase

VAR
	nHeadBoardType 	: USINT;
	nHeadNr			: SINT;		//Nummer des Heads (1 bzw -1 (untere Ebene)
	nParentSlotNr	: UINT;		//Head befindet sich zwar an keinem Slot, aber virtuell in der GUI (am Root)
	
	pFbZAxisRef		: POINTER TO FB_ZAxisRef;
	
	pCoHead			: POINTER TO FB_MzHead;
	pErrorChild 	: POINTER TO FB_MzTool;
	
	nStateA_InitAxisNext : USINT;
	
	pTempTool		: POINTER TO FB_MzTool;
	
	pExcludedTool	: POINTER TO FB_MzTool;
	
	pFlag			: BOOL;
	
	iterFlat		: FB_ObjCollectIterator;
	iterDeep		: FB_ObjCollectIteratorDeep;
	pDebugSlot		: POINTER TO FB_Slot;
	nDebugSlotNr	: UINT := 1;
END_VAR

VAR CONSTANT
	cNumberOfSlots : UINT := 7;
END_VAR

SUPER^();	//FB_MzBase aufrufen
pDebugSlot := fbSlotList.M_GetAtNr(nDebugSlotNr);

//Prozessdaten aktualisieren
stProcessData.n32Data[3] := REAL_TO_DINT(pXDrive^.P_rActPos);
stProcessData.n32Data[4] := REAL_TO_DINT(pYDrive^.P_rActPos);
stCurrentPos := P_stCurrentPosTotal;
stProcessData.n32Data[5] := REAL_TO_DINT(stCurrentPos.X);
stProcessData.n32Data[6] := REAL_TO_DINT(stCurrentPos.Y);
//ist nur für 2-Ebenen relevant
stProcessData.n32Data[7] := BOOL_TO_DINT(pYDrive^.P_bCoupled);

aObjProcData[nNotifyId] := stProcessData;

PROPERTY P_stCurrentPosPhys : ST_3DPoint
GET
VAR
	stTemp		: ST_3DPoint;
	stAbsPos : ST_3DPoint;
END_VAR
stAbsPos := P_stAbsPosPhys;
stTemp.X := pXDrive^.P_rActPos + stAbsPos.X;
stTemp.Y := pYDrive^.P_rActPos + stAbsPos.Y;
stTemp.Z := stAbsPos.Z;
P_stCurrentPosPhys := stTemp;
END_GET
END_PROPERTY

PROPERTY P_bCollFree : BOOL
GET
VAR
	pTool : POINTER TO FB_MzTool;
	iter : FB_ObjCollectIteratorDeep;
END_VAR
//Kollisionsfreihheit ist gegeben, wenn Unterkante Z-Wert von Tool >= kollissiongefährdete Höhe Workplate
IF nHeadNr < 0 THEN //unterer Head
	P_bCollFree := TRUE;
ELSE
	//alle ChildTools durchlaufen und checken, ob diese CollFree
	P_bCollFree := TRUE;
	pObjCollectNode^.nodes.M_GetIterator(iter);
	WHILE iter.pNode > 0 DO
		IF iter.pNode^.P_pObject > 0 and_then iter.pNode^.P_pObject^.M_bIsGroup(E_ObjectGroup.OBJECTGROUP_MzTool) THEN //schließt Pieces aus, da diese die Property 
			pTool := iter.pNode^.P_pObject;											//P_bCollFree nicht implementieren
			IF NOT pTool^.P_bCollFree THEN
				P_bCollFree := FALSE;
				RETURN;
			END_IF			
		END_IF
 	iter.M_Increment();
	END_WHILE	
END_IF
END_GET
END_PROPERTY

METHOD M_CheckChildsForActionBusy : BOOL
VAR_INPUT
	eAction : E_Action;
END_VAR
VAR
	pTool : POINTER TO FB_MzTool;
	iterDeep : FB_ObjCollectIteratorDeep;	
END_VAR
//Alle Childs durchlaufen
pObjCollectNode^.nodes.M_GetIterator(iterDeep);
WHILE iterDeep.pNode > 0 DO
	IF iterDeep.pNode^.P_pObject > 0 AND_THEN iterDeep.pNode^.P_pObject^.M_bIsGroup(E_ObjectGroup.OBJECTGROUP_MzTool) THEN
		pTool := iterDeep.pNode^.P_pObject;
		M_CheckChildsForActionBusy := pTool^.M_GetActionBusy(eAction);	
		IF M_CheckChildsForActionBusy THEN
			RETURN;
		END_IF
	END_IF
	iterDeep.M_Increment();
END_WHILE
END_METHOD

METHOD M_SetAllProps : ERRORID
VAR_INPUT
	refCmdData : REFERENCE TO  ST_CmdData;
END_VAR

VAR
	nNoOfYDrives : UINT;
	pDrive : POINTER TO FB_XYDriveBase;
	stHardwareID : ST_HardwareId;
END_VAR
M_SetAllProps := SUPER^.M_SetAllProps(refCmdData);
IF M_SetAllProps > 0 THEN
	RETURN;
END_IF

nParentSlotNr := DINT_TO_UINT(refCmdData.n32Data[1]);

nCurrentPropIndex := nCurrentPropIndex + 1;
nSpecPropIndex := nCurrentPropIndex;
nHeadNr := DINT_TO_SINT(refCmdData.n32Data[nCurrentPropIndex]);

nNoOfYDrives := fbXYDriveList.M_CountByGroup(E_HardwareGrp.AxisY);
IF nHeadNr = 1 AND nNoOfYDrives = 1 THEN //Normalfall für Plattform C
	stHardwareID.eGroup := E_HardwareGrp.AxisY;
	stHardwareID.nParentItem := 1;
	stHardwareID.nItem := 1;
	pDrive := fbXYDriveList.M_GetByHwId(stHardwareID);
	IF pDrive > 0 THEN
		pYDrive := pDrive;
	ELSE
		M_SetAllProps := E_ErrorIdObjMgmt.ERRORID_InvalidHardwareRef;
		RETURN;
	END_IF
ELSIF nHeadNr = 1 AND nNoOfYDrives = 2 THEN //Plattform D oberer Head
	stHardwareID.eGroup := E_HardwareGrp.AxisY;
	stHardwareID.nParentItem := 1;
	stHardwareID.nItem := 2;
	pDrive := fbXYDriveList.M_GetByHwId(stHardwareID);
	IF pDrive > 0 THEN
		pYDrive := pDrive;
	ELSE
		M_SetAllProps := E_ErrorIdObjMgmt.ERRORID_InvalidHardwareRef;
		RETURN;
	END_IF	
	
ELSIF nHeadNr = -1 AND nNoOfYDrives = 2 THEN //Plattform D unterer Head
	stHardwareID.eGroup := E_HardwareGrp.AxisY;
	stHardwareID.nParentItem := 1;
	stHardwareID.nItem := 1;
	pDrive := fbXYDriveList.M_GetByHwId(stHardwareID);
	IF pDrive > 0 THEN
		pYDrive := pDrive;
	ELSE
		M_SetAllProps := E_ErrorIdObjMgmt.ERRORID_InvalidHardwareRef;
		RETURN;
	END_IF
ELSE
	M_SetAllProps := E_ErrorIdObjMgmt.ERRORID_InvalidMultiZNr;
	RETURN;
END_IF

pFbMultiZ := pDrive^.P_pMultiZRef;

//X
stHardwareID.eGroup := E_HardwareGrp.AxisX;
stHardwareID.nParentItem := 0;
stHardwareID.nItem := 1;
pDrive := fbXYDriveList.M_GetByHwId(stHardwareID);
IF pDrive > 0 THEN
	pXDrive := pDrive;
ELSE
	M_SetAllProps := E_ErrorIdObjMgmt.ERRORID_InvalidHardwareRef;
	RETURN;
END_IF

//Type der ZBasis-Platine (derzeit nur 0 oder 1)
//0= keine BasisPlatine vorhanden, es können auch keine Achsen betrieben werden
//1= BasisPlatine vorhanden
nCurrentPropIndex := nCurrentPropIndex + 1;
nHeadBoardType := DINT_TO_USINT(refCmdData.n32Data[nCurrentPropIndex]);
IF NOT (nHeadBoardType >= 0 AND nHeadBoardType <= 1) THEN
	M_SetAllProps := E_ErrorIdObjMgmt.ERRORID_InvalidHeadBoardType;
	RETURN;	
END_IF

IF nHeadBoardType = 1 AND pFbMultiZ = 0 THEN
	M_SetAllProps := E_ErrorIdObjMgmt.ERRORID_HeadBoardNotAvailable;
	RETURN;		
END_IF

nNoOfProps := nCurrentPropIndex + 1;
END_METHOD

METHOD M_CheckMoveLimit : BOOL
VAR_INPUT
	sAxis			: STRING[2];
	eMoveMode		: E_MoveMode;
	rMovePosition	: REAL;
END_VAR

VAR
	st3DPoint		: ST_3DPoint;
	rMovePosTemp	: REAL;
END_VAR
IF sAxis = 'Z' THEN //Head gibt in "Z" immer TRUE zurück, da er sich in Z nicht bewegt
	M_CheckMoveLimit := TRUE;
ELSE
	M_CheckMoveLimit := SUPER^.M_CheckMoveLimit(sAxis,eMoveMode,rMovePosition);
END_IF
END_METHOD

METHOD M_ClearAllProps
VAR_INPUT
	bIgnoreParent : BOOL; //Es wird das gesamte OD gelöscht. -> Zeiger auf Parent nicht mehr gültig!
END_VAR
nHeadNr := 0;
SUPER^.M_ClearAllProps(bIgnoreParent);
END_METHOD

PROPERTY P_bZIsMoving : BOOL
SET
END_SET
GET
VAR
	iter : FB_ObjCollectIteratorDeep;
	pTool : POINTER TO FB_MzTool;
	bTemp : BOOL;
END_VAR
pObjCollectNode^.nodes.M_GetIterator(iter);
WHILE iter.pNode > 0 DO
	IF iter.pNode^.P_pObject > 0 AND_THEN iter.pNode^.P_pObject^.M_bIsGroup(E_ObjectGroup.OBJECTGROUP_MzTool) THEN
		pTool := iter.pNode^.P_pObject;
		IF pTool^.P_bZIsMoving THEN
			bTemp := TRUE;
			EXIT;
		END_IF
	END_IF
	iter.M_Increment();
END_WHILE
P_bZIsMoving:= bZIsMoving OR bTemp;
END_GET
END_PROPERTY

METHOD FB_init : BOOL
VAR_INPUT
	bInitRetains : BOOL; // if TRUE, the retain variables are initialized (warm start / cold start)
	bInCopyCode : BOOL;  // if TRUE, the instance afterwards gets moved into the copy code (online change)
END_VAR
eObjectType := E_ObjectType.OBJECTTYPE_MZHead;
eObjectGroup := E_ObjectGroup.OBJECTGROUP_MzTool OR E_ObjectGroup.OBJECTGROUP_Device;
END_METHOD

METHOD M_GetMinMaxActPos
VAR_INPUT
	pData : POINTER TO ARRAY[0..19] OF DINT;
END_VAR
VAR
	stCurrPosTotal : ST_3DPoint;
END_VAR
SUPER^.M_GetMinMaxActPos(pData);

stCurrPosTotal := P_stCurrentPosTotal;
pData^[6] := REAL_TO_DINT(stCurrPosTotal.X);
pData^[7] := REAL_TO_DINT(stCurrPosTotal.Y);
pData^[8] := REAL_TO_DINT(stCurrPosTotal.Z);
END_METHOD

PROPERTY P_bIsInit : BOOL
GET
P_bIsInit := bInitAxisOk AND pXDrive^.P_bHomed AND pYDrive^.P_bHomed;
END_GET
END_PROPERTY

PROPERTY P_stAbsPosPhys : ST_3DPoint
GET
VAR
	stTemp	: ST_3DPoint;
END_VAR
//X und Y beziehen sich auf den Koordinatenursprung, wenn die Achsen theoretischn aus Antrieb (0;0) stehen
P_stAbsPosPhys := F_Add3DPoints(stRelPos,stOffset);
END_GET
END_PROPERTY

PROPERTY P_nParentSlotNr : UINT
GET
P_nParentSlotNr := nParentSlotNr;
END_GET
END_PROPERTY

PROPERTY P_bHasZSensorSlot : BOOL
GET
P_bHasZSensorSlot := TRUE;
END_GET
END_PROPERTY

ACTION A_Init:
stError.POUState := nStateA_InitAxis;

CASE nStateA_InitAxis OF
	0:
		bInitAxisOk := FALSE;
		bInitReadyX := FALSE;
		bInitReadyY := FALSE;
		bInitErrorX := FALSE;
		bInitErrorY := FALSE;
		nStateA_InitAxis := 1;
		nCurInitZAxis := 0;

		IF nHeadBoardType = 0 THEN	//Head besitzt keine HeadBoard und somit auch keine Z-Achsen		
			nStateA_InitAxis := 4;	//weiter zum Dispacher
		END_IF
		
	1:	//ALLE Z-Achsen die noch nicht zur Initalisierung durch andere Tools angestoßen wurde, initialisieren
		nCurInitZAxis := nCurInitZAxis + 1;	
		FOR i := nCurInitZAxis TO 7 BY 1 DO
			//Ist Achse auch physikalisch vorhanden und ist sie keine SubAchse (wird von Stamp gesteuert)
			pFbZAxisRef := ADR(pFbMultiZ^.aFbZAxisRef[i]);
			IF pFbZAxisRef^.stInput.nStatus.7 AND NOT pFbZAxisRef^.bIsSubAxis THEN
				IF (NOT pFbZAxisRef^.stStatus.bIsHoming AND NOT pFbZAxisRef^.stStatus.bIsHomed)
					OR (NOT pFbZAxisRef^.stStatus.bIsHoming AND (pFbZAxisRef^.P_rHomePos - pFbZAxisRef^.P_rCurrentPos) > 20) THEN
					nCurInitZAxis := UINT_TO_USINT(i);
					nStateA_InitAxis := 2; //Init Z-Achse anstoßen
					fbZmHome(bExecute:= TRUE, pFbZAxisRef:= pFbZAxisRef, bMoveToHome:= TRUE);
					RETURN;
				ELSE
					IF nCurInitZAxis = 7 THEN
						nStateA_InitAxis := 3;	//weiter zu Check eigene Tools
					END_IF
				END_IF
			ELSE
				IF nCurInitZAxis = 7 THEN
					nStateA_InitAxis := 3;	//weiter zu Check eigene Tools
				END_IF				
			END_IF
		END_FOR
		
	2:	//Z-Achse initialisieren
		fbZmHome(bExecute:= TRUE, pFbZAxisRef:= pFbZAxisRef, bMoveToHome:= TRUE);
		IF NOT fbZmHome.bBusy THEN
			IF fbZmHome.bError THEN
				stError.ErrorId := fbZmHome.nErrorId;
				stError.HardwareGrp := E_HardwareGrp.AxisZ;
				stError.HardwareNr	:= nCurInitZAxis;
				nStateA_InitAxis := 99;
			ELSE
				IF nCurInitZAxis = 7 THEN
					nStateA_InitAxis := 3;	//weiter zu check
				ELSE
					nStateA_InitAxis := 1;	//nächste Z-Achse
				END_IF
			END_IF
			fbZmHome(bExecute:= FALSE);
		END_IF
		
	3:	//alle eigenen Tools auf Fehlerfreiheit checken
		IF P_bNoChildBusy THEN
			pErrorChild := M_GetFirstErrorChild(FALSE);
			IF pErrorChild > 0 THEN
				stError.ErrorId := pErrorChild^.P_nErrorId;
				nStateA_InitAxis := 99;
			ELSE
				//Test CrashSafe
				IF P_bCollFree THEN
					nStateA_InitAxis := 4;
				ELSE
					stError.ErrorId := E_ErrorIdCmd.ERRORID_AnyToolNotCrashSafe;
					stError.HardwareGrp := E_HardwareGrp.AxisZ;
					nStateA_InitAxis := 99;
				END_IF
			END_IF
		END_IF

	4:	//Dispacher!!!!!!!!!!!!!!!!!!!!
		IF nHeadNr = 1 THEN  //oberer Head
			IF pXDrive^.P_bHoming THEN //X-bereits homing -> Y-Homing
				//kein weiterer Check notwendig
				nStateA_InitAxis := 20;	//Y-Homing
				nStateA_InitAxisNext := 40;
			ELSE //XY-Homing
				//falls es einen unteren Head gibt, muss dieser auch sicher sein
				IF pCoHead > 0 THEN
					IF pCoHead^.P_bNoChildBusy THEN
						pErrorChild := pCoHead^.M_GetFirstErrorChild(FALSE);
						IF pErrorChild > 0 THEN
							stError.ErrorId := pErrorChild^.P_nErrorId;
							nStateA_InitAxis := 99;
						ELSE
							//Test CrashSafety
							IF pCoHead^.P_bCollFree THEN
								nStateA_InitAxis := 30;
								nStateA_InitAxisNext := 40;
							ELSE
								stError.ErrorId := E_ErrorIdCmd.ERRORID_AnyToolNotCrashSafe;
								stError.HardwareGrp := E_HardwareGrp.AxisZ;
								nStateA_InitAxis := 99;
							END_IF
						END_IF
					END_IF
				END_IF
				nStateA_InitAxis := 30; //XY-Homing
				nStateA_InitAxisNext := 40;
			END_IF
		ELSIF nHeadNr = -1 THEN  //unterer Head
			IF pXDrive^.P_bHoming THEN  //X-bereits homing und homingzeit > 3s -> Y-Homing
				//Abfrage Zeit???
				IF pXDrive^.P_tHomingTime >= T#3S THEN
					nStateA_InitAxis := 20;	//Y-Homing
					nStateA_InitAxisNext := 40;
				END_IF
			ELSE
				IF pXDrive^.P_bHomed THEN
					IF (pXDrive^.P_rActPos > pXDrive^.P_rMinPos) THEN
						nStateA_InitAxis := 20;	//Y-Homing
						nStateA_InitAxisNext := 40;
					END_IF
				ELSE
					//Oberer Head ChrashSafety?
					IF pCoHead^.P_bCollFree THEN
						//zuerst X-Homing anstoßen und nach 5s Y-Homing anstoßen
						nStateA_InitAxis := 10;	//X-Homing
						nStateA_InitAxisNext := 5;
					END_IF
				END_IF
			END_IF
		END_IF
		
	5:	//Waiting bis X-Homing aktiv - Dieser Schritt wird nur für unteren Head benötigt
		IF pXDrive^.P_tHomingTime > T#0S THEN
			nStateA_InitAxis := 4; //zurück zum Dispacher
		END_IF
		
	10:	//X-Homing
		nStateA_InitAxis := nStateA_InitAxisNext;
		IF NOT pXDrive^.P_bHoming THEN
			stError.ErrorId := pXDrive^.M_Init(bReInit);	
		END_IF
		IF stError.ErrorId > 0 THEN
			nStateA_InitAxis := 99;
		END_IF
	
	20:	//Y-Homing
		nStateA_InitAxis := nStateA_InitAxisNext;
		stError.ErrorId := pYDrive^.M_Init(bReInit);
		IF stError.ErrorId > 0 THEN
			nStateA_InitAxis := 99;
		END_IF
	
	30:	//XY-Homing
		nStateA_InitAxis := nStateA_InitAxisNext;
		IF NOT pXDrive^.P_bHoming THEN
			stError.ErrorId := pXDrive^.M_Init(bReInit);	
		END_IF
		IF stError.ErrorId > 0 THEN
			nStateA_InitAxis := 99;
		ELSE
			stError.ErrorId := pYDrive^.M_Init(bReInit);
		END_IF
		
	40:	//XY-Homing ready?
		IF NOT pXDrive^.P_bBusy THEN
			IF pXDrive^.P_bError THEN
				stError.ErrorId := pXDrive^.P_nErrorId;
				stError.HardwareGrp := E_HardwareGrp.AxisX;
				stError.HardwareNr	:= 1;
				IF pYDrive^.P_bBusy THEN
					pYDrive^.M_Stop();	
				END_IF
				bInitErrorX := TRUE;
			ELSE
				bInitReadyX := TRUE;
			END_IF
		END_IF

		IF NOT pYDrive^.P_bBusy THEN
			IF pYDrive^.P_bError THEN
				stError.ErrorId := pYDrive^.P_nErrorId;
				stError.HardwareGrp := E_HardwareGrp.AxisY;
				stError.HardwareNr	:= 1;
				IF pXDrive^.P_bBusy THEN
					pXDrive^.M_Stop();	
				END_IF
				bInitErrorY := TRUE;
			ELSE
				bInitReadyY := TRUE;
			END_IF
		END_IF

		IF bInitReadyX AND bInitReadyY THEN	//beide Achsen ohne Fehler initialisiert
			bInitAxisOk := TRUE;
			nStateA_InitAxis := 80;
		ELSIF (bInitReadyX AND bInitErrorY) OR (bInitErrorX AND bInitReadyY) OR (bInitErrorX AND bInitErrorY) THEN //mind. 1 Achse in Fehler
			//Problem: wenn beide Achsen in Fehler gehen, dann wird nur die zweite als Fehler angezeigt?
			stError.POUState := nStateA_InitAxis;
			nStateA_InitAxis := 99;
		END_IF

	70:	//Abbrechen
		//Die Initialisierung der Z-Achsen lässt sich nicht stoppen
		fbZmHome(bExecute:= FALSE);
		
		//Die XY-Achsen können gestoppt werden
		IF pXDrive^.P_bBusy THEN
			pXDrive^.M_Stop();	
		END_IF
		
		IF pYDrive^.P_bBusy THEN
			pYDrive^.M_Stop();	
		END_IF

		IF NOT (pXDrive^.P_bBusy OR pYDrive^.P_bBusy) THEN
			bInitReadyX := FALSE;
			bInitReadyY := FALSE;
			bInitErrorX := FALSE;
			bInitErrorY := FALSE;
			nStateA_InitAxis := 80;
		END_IF	
END_CASE

//Errorhandling
IF nStateA_InitAxis = 99 THEN
	bInitErrorX := FALSE;
	bInitErrorY := FALSE;
	stError.ObjectId := nObjectID;
	stError.Cmd := E_Action.ACTION_Init;
	stError.POU := E_POU.POU_FB_MzHead;
	stError.POUAction := E_POUACT.POUACT_A_Init;
	fbErrorList.M_Add(stError);
END_IF
END_ACTION

METHOD M_CheckAction : ERRORID
VAR_INPUT
	refActionData 	: REFERENCE TO ST_ActionData;
	pCorrelObject	: POINTER TO FB_Object;
END_VAR
IF refActionData.eAction = E_Action.ACTION_MoveToTarget THEN
	//Diese Action wird nur für den unteren Head benötigt, wenn er keine Z-Achsen hat. (Collimator)
	//Es erfolgt keine Z-Zustellung.
	RETURN;
ELSE
	M_CheckAction := SUPER^.M_CheckAction(refActionData,pCorrelObject);
END_IF
END_METHOD

METHOD M_GetCollFree : BOOL
VAR_INPUT
	rDistanceX : REAL;
	rDistanceY : REAL;
END_VAR

VAR
	pTool : POINTER TO FB_MzTool;
	iter : FB_ObjCollectIteratorDeep;
END_VAR
//Ermittlung, ob anhängende Tools in kollisionsfreiem Bereich
//Kollisionsfreihheit ist gegeben, wenn Unterkante Z-Wert von Tool >= kollissiongefährdete Höhe Workplate
IF P_bIsTopHead THEN
	//alle ChildTools durchlaufen und checken, ob diese CollFree
	M_GetCollFree := TRUE;
	pObjCollectNode^.nodes.M_GetIterator(iter);
	WHILE iter.pNode > 0 AND_THEN iter.pNode^.P_pObject > 0 DO
		IF iter.pNode^.P_pObject^.M_bIsGroup(E_ObjectGroup.OBJECTGROUP_MzTool) THEN
			pTool := iter.pNode^.P_pObject;
			IF NOT pTool^.M_GetCollFree(rDistanceX,rDistanceY) THEN
				M_GetCollFree := FALSE;
				RETURN;
			END_IF			
		END_IF	
		iter.M_Increment();
	END_WHILE	
ELSE
	 M_GetCollFree := TRUE;
END_IF
END_METHOD

METHOD M_ExeAction : ERRORID
VAR_INPUT
	refActionData : REFERENCE TO ST_ActionData;	
END_VAR
IF NOT (eCurrentState = E_MachineState.MACHINESTATE_Idle OR
	eCurrentState = E_MachineState.MACHINESTATE_Active OR
	eCurrentState = E_MachineState.MACHINESTATE_Ready) THEN
	M_ExeAction := E_ErrorIdCmd.ERRORID_InvalidState;
	RETURN;
END_IF

CASE refActionData.eAction OF
	
	E_Action.ACTION_MoveZ:
		IF NOT bMoveZ THEN
			//Dient nur zum freifahren aller Tools die, an diesem Head hängen	
			eMoveModeZ := DINT_TO_USINT(refActionData.aParams[1]);
			
			//Head darf nur alle in ihm hängende Tools freifahren oder auf "0" fahren
			IF NOT (eMoveModeZ = E_MoveMode.MODE_Free OR eMoveModeZ = E_MoveMode.MODE_Home) THEN
				M_ExeAction := E_ErrorIdCmd.ERRORID_InvalidMoveMode;
				RETURN;
			END_IF
			
			bZIsMoving := TRUE;
			bMoveZ := TRUE;			
			fbList.A_AddHeadValue(hList := hList, putValue := E_Action.ACTION_MoveZ);
			
		ELSE
			M_ExeAction := E_ErrorIdCmd.ERRORID_BasicActionActive;  //Error
			RETURN;				
		END_IF	

	ELSE
		M_ExeAction := SUPER^.M_ExeAction(refActionData);
		RETURN;
END_CASE
bBusy := TRUE;
eCurrentState := E_MachineState.MACHINESTATE_Active;
END_METHOD

PROPERTY P_bIsTopHead : BOOL
GET
IF nHeadNr = 1 THEN	// Besagt, dass es ein oberer Head ist.
	P_bIsTopHead := TRUE;
END_IF
END_GET
END_PROPERTY

PROPERTY P_pCoHead : POINTER TO FB_MzHead
GET
P_pCoHead := pCoHead;
END_GET
END_PROPERTY

PROPERTY P_bIsHot : BOOL
GET
VAR
	pTool : POINTER TO FB_MzTool;
	iter : FB_ObjCollectIteratorDeep;
END_VAR
//Alle Childs durchlaufen
pObjCollectNode^.nodes.M_GetIterator(iter);
WHILE iter.pNode > 0 AND_THEN iter.pNode^.P_pObject > 0 DO
	IF iter.pNode^.P_pObject^.M_bIsGroup(E_ObjectGroup.OBJECTGROUP_MzTool) THEN
		pTool := iter.pNode^.P_pObject;
		IF pTool^.P_bIsHot THEN
			P_bIsHot := TRUE;
			RETURN;
		END_IF
	END_IF
	iter.M_Increment();
END_WHILE
END_GET
END_PROPERTY

METHOD M_CheckChildsForError : ERRORID
VAR_INPUT
END_VAR
VAR
	pTool : POINTER TO FB_MzTool;
	iterDeep : FB_ObjCollectIteratorDeep;	
END_VAR
//Alle Childs durchlaufen
pObjCollectNode^.nodes.M_GetIterator(iterDeep);
WHILE iterDeep.pNode > 0 DO
	IF iterDeep.pNode^.P_pObject > 0 AND_THEN iterDeep.pNode^.P_pObject^.M_bIsGroup(E_ObjectGroup.OBJECTGROUP_MzTool) THEN
		pTool := iterDeep.pNode^.P_pObject;
		M_CheckChildsForError := pTool^.P_nErrorId;
		IF M_CheckChildsForError > 0 THEN
			RETURN;			
		END_IF
	END_IF
	iterDeep.M_Increment();
END_WHILE
END_METHOD

PROPERTY P_rMaxCollFreeHeight : REAL
GET
VAR
	pTool	: POINTER TO FB_MzTool;
	iter : FB_ObjCollectIteratorDeep;
	stPos	: ST_3DPoint;
END_VAR
stPos := P_stAbsPosPhys;
P_rMaxCollFreeHeight := stPos.Z;
pObjCollectNode^.nodes.M_GetIterator(iter);
WHILE iter.pNode > 0 DO
	IF iter.pNode^.P_pObject > 0 AND_THEN iter.pNode^.P_pObject^.M_bIsGroup(E_ObjectGroup.OBJECTGROUP_MzTool) THEN
		pTool := iter.pNode^.P_pObject;
		stPos := pTool^.P_stAbsPosTotal;
		stPos.Z := stPos.Z + pTool^.P_pZAxisRef^.P_rMaxPos;
		IF stPos.Z < P_rMaxCollFreeHeight THEN
			P_rMaxCollFreeHeight := stPos.Z;
		END_IF
	END_IF
	iter.M_Increment();
END_WHILE
END_GET
END_PROPERTY

METHOD M_GetAllProps : ERRORID
VAR_INPUT
	refCmdData : REFERENCE TO  ST_CmdData;
END_VAR
//Basisproperties lesen
SUPER^.M_GetAllProps(refCmdData);

refCmdData.n32Data[1] := nParentSlotNr;

//Specialproperties lesen
nCurrentPropIndex := nCurrentPropIndex + 1;
refCmdData.n32Data[nCurrentPropIndex] := nHeadNr;
nCurrentPropIndex := nCurrentPropIndex + 1;
refCmdData.n32Data[nCurrentPropIndex] := nHeadBoardType;
END_METHOD

PROPERTY P_bNoChildBusy : BOOL
GET
VAR
	pTool : POINTER TO FB_MzTool;
	iter : FB_ObjCollectIteratorDeep;
END_VAR
P_bNoChildBusy := TRUE;
pObjCollectNode^.nodes.M_GetIterator(iter);
WHILE iter.pNode > 0 DO
	IF iter.pNode^.P_pObject > 0 AND_THEN iter.pNode^.P_pObject^.M_bIsGroup(E_ObjectGroup.OBJECTGROUP_MzTool) THEN
		pTool := iter.pNode^.P_pObject;
		IF pTool^.P_bBusy THEN
			P_bNoChildBusy := FALSE;
			RETURN;
		END_IF
	END_IF
	iter.M_Increment();
END_WHILE
END_GET
END_PROPERTY

METHOD M_AddChild : ERRORID
VAR_INPUT
	pObject : POINTER TO FB_Object;
	nSlotNr	: UINT;
	nIndex 	: INT;
END_VAR

VAR
	pSlot : POINTER TO FB_Slot;
END_VAR
//Mögliche Childs sind nur MzTools
//muss unbedingt an ein Slot (in diesem Fall die Achse)
IF pObject > 0 AND_THEN pObject^.M_bIsGroup(E_ObjectGroup.OBJECTGROUP_MzTool) THEN
	//Slot holen
	pSlot := fbSlotList.M_GetAtNr(nSlotNr);
	IF pSlot > 0 THEN
		IF pSlot^.P_pChild = 0 THEN
			//Object darf selber noch an keinem Parent hängen
			IF pObject^.P_pParentObject = 0 THEN
				pSlot^.P_pChild := pObject;
				pObject^.P_pObjCollectNode := pObjCollectNode^.nodes.M_AddNewNode(pObject,nIndex);
				pObject^.M_UpdateParent();
			ELSE
				M_AddChild := E_ErrorIdObjMgmt.ERRORID_ObjectAlreadyOnAnotherParent;
			END_IF
		ELSE //Slot bereits belegt
			M_AddChild := E_ErrorIdObjMgmt.ERRORID_SlotIsAlreadyOccupied;
		END_IF
	ELSE
		M_AddChild := E_ErrorIdObjMgmt.ERRORID_InvalidSlotNumber;	
	END_IF
ELSE
	M_AddChild := E_ErrorIdObjMgmt.ERRORID_InvalidObject;
END_IF
END_METHOD

ACTION A_Reset:
nStateA_ResetTool := 80;
SUPER^.A_Reset();
END_ACTION

PROPERTY P_bXYIsMoving : BOOL
GET
VAR
	iter : FB_ObjCollectIteratorDeep;
	pTool : POINTER TO FB_MzTool;
	bTemp : BOOL;
END_VAR
pObjCollectNode^.nodes.M_GetIterator(iter);
WHILE iter.pNode > 0 DO
	IF iter.pNode^.P_pObject > 0 AND_THEN iter.pNode^.P_pObject^.M_bIsGroup(E_ObjectGroup.OBJECTGROUP_MzTool) THEN
		pTool := iter.pNode^.P_pObject;
		IF pTool^.P_bXYIsMoving THEN
			bTemp := TRUE;
			EXIT;
		END_IF
	END_IF
	iter.M_Increment();
END_WHILE
P_bXYIsMoving:= bXYIsMoving OR bTemp;
END_GET
SET
bXYIsMoving := P_bXYIsMoving;
END_SET
END_PROPERTY

METHOD M_CheckProps : ERRORID
VAR_INPUT
END_VAR
M_CheckProps := SUPER^.M_CheckProps();
IF M_CheckProps > 0 THEN
	RETURN;
END_IF

IF nHeadNr > 0 THEN	//oben
	IF stRelPos.Z < 40000 THEN
		M_CheckProps := E_ErrorIdObjMgmt.ERRORID_InvalidRelPosZ;
		RETURN;
	END_IF
ELSIF nHeadNr < 0 THEN	//unten
	IF stRelPos.Z > -200000 THEN
		M_CheckProps := E_ErrorIdObjMgmt.ERRORID_InvalidRelPosZ;
		RETURN;
	END_IF
END_IF

pCoHead := fbObjectDirectory.M_GetCoHead(THIS);

IF afbWorkplate[1].P_nObjectID > 0 THEN
	pAssignWorkplate := ADR(afbWorkplate[1]); 
ELSE
	M_CheckProps := E_ErrorIdObjMgmt.ERRORID_NoWorkplateCreated;
END_IF
END_METHOD

ACTION A_MoveZ:
CASE nStateA_MoveZ OF
	0:	//Tools ermitteln, bei denen nReducedDist gesetzt ist und diese freifahren
		//das sind die Tools, die durch Dock in einem Target bzw. Piece eingeführt sind und wieder langsam herausgefahren
		//werden müssen
		stActionData.eAction := E_Action.ACTION_MoveZ;
		stActionData.aParams[1] := eMoveModeZ;
		stActionData.aParams[3] := -1; //Max Speed
	
		nStateA_MoveZ := 2;
		pObjCollectNode^.nodes.M_GetIterator(iterDeep);
		WHILE iterDeep.pNode > 0 DO
			IF iterDeep.pNode^.P_pObject > 0 AND_THEN iterDeep.pNode^.P_pObject^.M_bIsGroup(E_ObjectGroup.OBJECTGROUP_MzTool) THEN
				pTempTool := iterDeep.pNode^.P_pObject;
				IF pTempTool^.P_nReducedMoveZDist <> 0 THEN
					IF NOT pTempTool^.P_bIsInit THEN
						stError.ErrorId := E_ErrorIdCmd.ERRORID_DeviceNotInitialized;
						stError.POUState := nStateA_MoveZ;
						nStateA_MoveZ := 99;
						EXIT;
					ELSE
						IF (NOT pTempTool^.P_bCollFree) OR (eMoveModeZ = E_MoveMode.MODE_Home) THEN
							stError.ErrorId := pTempTool^.M_ExeAction(stActionData);
							IF stError.ErrorId > 0 THEN
								stError.POUState := nStateA_MoveZ;
								nStateA_MoveZ := 99;
								EXIT;
							ELSE
								nStateA_MoveZ := 1;	
							END_IF
						END_IF					
					END_IF
				END_IF
			END_IF
			iterDeep.M_Increment();
		END_WHILE
		
	1:	//warten, bis diese Tools fertig
		nStateA_MoveZ := 2;
		pObjCollectNode^.nodes.M_GetIterator(iterDeep);
		WHILE iterDeep.pNode > 0 DO
			IF iterDeep.pNode^.P_pObject > 0 AND_THEN iterDeep.pNode^.P_pObject^.M_bIsGroup(E_ObjectGroup.OBJECTGROUP_MzTool) THEN
				pTempTool := iterDeep.pNode^.P_pObject;
				IF pTempTool^.P_bError THEN
					stError.POUState := nStateA_MoveZ;
					nStateA_MoveZ := 99;
					EXIT;
				ELSE
					IF pTempTool^.M_GetActionBusy(E_Action.ACTION_MoveZ) THEN
						nStateA_MoveZ := 1;
					END_IF
				END_IF
			END_IF
			iterDeep.M_Increment();
		END_WHILE
		
	2:	//auf alle Tools anwenden
		//neu! pro Achse nur noch das Tool freifahren, welches am nächsten zur Workplate befindet
		stActionData.eAction := E_Action.ACTION_MoveZ;
		stActionData.aParams[1] := eMoveModeZ;
		stActionData.aParams[3] := -1; //Max Speed
		nStateA_MoveZ := 80;
		//nicht mehr alle Tools durchlaufen, sondern nur noch die direkten Childs an den Achsen
		pObjCollectNode^.nodes.M_GetIterator(iterFlat);
		WHILE iterFlat.pNode > 0 DO
			IF iterFlat.pNode^.P_pObject > 0 AND_THEN iterFlat.pNode^.P_pObject^.M_bIsGroup(E_ObjectGroup.OBJECTGROUP_MzTool) THEN
				//Hier steht das obers Tool, welches sich an der Achse befinder zur Verfügung
				pFlag := FALSE;
				pTempTool := iterFlat.pNode^.P_pObject;
				pTempTool := pTempTool^.M_GetClosestTool(FALSE);
				IF pExcludedTool > 0 THEN				
					//Falls sich pTempTool auf der gleichen Achse wie pExcluded Tool befindet, dann dieses auch auschließen
					IF pTempTool^.P_nZAxisNr <> pExcludedTool^.P_nZAxisNr THEN
						pFlag := TRUE;
					END_IF					
				ELSE
					pFlag := TRUE;
				END_IF
				
				IF pFlag THEN
					IF NOT pTempTool^.P_bIsInit THEN
						stError.ErrorId := E_ErrorIdCmd.ERRORID_DeviceNotInitialized;
						stError.POUState := nStateA_MoveZ;
						nStateA_MoveZ := 99;
						EXIT;
					ELSE
						IF (NOT pTempTool^.P_bCollFree) OR (eMoveModeZ = E_MoveMode.MODE_Home) THEN
							stError.ErrorId := pTempTool^.M_ExeAction(stActionData);
							IF stError.ErrorId > 0 THEN
								stError.POUState := nStateA_MoveZ;
								nStateA_MoveZ := 99;
								EXIT;
							ELSE
								nStateA_MoveZ := 3;	
							END_IF
						END_IF
					END_IF
				END_IF				
				
			END_IF
			iterFlat.M_Increment();
		END_WHILE
		
		pExcludedTool := 0;
	
	3:	//warten bis alle Tools fertig
		nStateA_MoveZ := 80;
		pObjCollectNode^.nodes.M_GetIterator(iterDeep);
		WHILE iterDeep.pNode > 0 DO
			IF iterDeep.pNode^.P_pObject > 0 AND_THEN iterDeep.pNode^.P_pObject^.M_bIsGroup(E_ObjectGroup.OBJECTGROUP_MzTool) THEN
				pTempTool := iterDeep.pNode^.P_pObject;
				IF pTempTool^.P_bError THEN
					stError.POUState := nStateA_MoveZ;
					nStateA_MoveZ := 99;
					EXIT;
				ELSE
					IF pTempTool^.M_GetActionBusy(E_Action.ACTION_MoveZ) THEN
						nStateA_MoveZ := 3;
					END_IF
				END_IF
			END_IF
			iterDeep.M_Increment();
		END_WHILE
		
	70:	//Stoppen
		pObjCollectNode^.nodes.M_GetIterator(iterDeep);
		WHILE iterDeep.pNode > 0 DO
			IF iterDeep.pNode^.P_pObject > 0 AND_THEN iterDeep.pNode^.P_pObject^.M_bIsGroup(E_ObjectGroup.OBJECTGROUP_MzTool) THEN
				pTempTool := iterDeep.pNode^.P_pObject;
				pTempTool^.M_CancelAction(E_ACTION.ACTION_MoveZ);
			END_IF
			iterDeep.M_Increment();
		END_WHILE
		nStateA_MoveZ := 71;
		
	71: //Alles Tools ready?
		nStateA_MoveZ := 80;
		pObjCollectNode^.nodes.M_GetIterator(iterDeep);
		WHILE iterDeep.pNode > 0 DO
			IF iterDeep.pNode^.P_pObject > 0 AND_THEN iterDeep.pNode^.P_pObject^.M_bIsGroup(E_ObjectGroup.OBJECTGROUP_MzTool) THEN
				pTempTool := iterDeep.pNode^.P_pObject;
				IF pTempTool^.P_bError THEN
					stError.POUState := nStateA_MoveZ;
					nStateA_MoveZ := 99;
					EXIT;
				ELSE
					IF pTempTool^.M_GetActionBusy(E_Action.ACTION_MoveZ) THEN
						nStateA_MoveZ := 71;
					END_IF
				END_IF
			END_IF
			iterDeep.M_Increment();
		END_WHILE
END_CASE

//Errorhandling
IF nStateA_MoveZ = 99 THEN
	stError.ObjectId := nObjectID;
	stError.Cmd := E_Action.ACTION_MoveZ;
	stError.POU := E_POU.POU_FB_MzHead;
	stError.POUAction := E_POUACT.POUACT_A_MoveZ;
	fbErrorList.M_Add(stError);
END_IF
END_ACTION

METHOD M_GetZAxisRef : POINTER TO FB_ZAxisRef
VAR_INPUT
	pTool : POINTER TO FB_MzTool;
	pToolSlot : POINTER TO FB_Slot;
END_VAR
IF pToolSlot > 0 THEN
	M_GetZAxisRef := ADR(pFbMultiZ^.aFbZAxisRef[pToolSlot^.P_nNr]);
END_IF
END_METHOD

METHOD M_MoveFree : ERRORID
VAR_INPUT
	pExcludedTool : POINTER TO FB_MzTool;
END_VAR
stActionData.eAction := E_Action.ACTION_MoveZ;
stActionData.aParams[1] := E_MoveMode.MODE_Free;
THIS^.pExcludedTool := pExcludedTool;
M_MoveFree := M_ExeAction(stActionData);
END_METHOD

PROPERTY P_pMzHead : POINTER TO FB_MzHead
GET
P_pMzHead := THIS;
END_GET
END_PROPERTY

END_FUNCTION_BLOCK

// ---- Objects/Targets/Active/FB_CustomUnitType1.TcPOU
FUNCTION_BLOCK FB_CustomUnitType1 EXTENDS FB_ActiveTarget IMPLEMENTS I_SlotTarget
VAR
	
	fbSlotList			: FB_SlotList;
	pSlot				: POINTER TO FB_DimSlot;
	nNumberOfSlots		: UINT;
	nFirstSlotPropIndex	: UINT;	//erster Index für Slots (benötigt in M_SetSingleProps)
	nLastSlotPropIndex	: UINT;	//letzte Index für Slots (benötigt in M_SetSingleProps)
	
	//Spec-Properties
	nValveNrSlot1		: USINT;
	nValveNrSlot2		: USINT;
	nPumpNrWaste		: USINT;
	nBottleNrWaste 		: USINT;
	
	//****************************************Aktionvariablen****************************************************
	
	//Action: "SuckOff"
	bSuckOff			: BOOL;
	nStateA_SuckOff		: USINT;
	nSuckOffChannel		: USINT;
	bSuckOff_On			: BOOL;
	tTime				: TIME;
	tmrTime				: TON;
	tDelayValveOff		: TIME;
	tmrDelayValveOff	: TON;
	
	
END_VAR

IF bInitFB THEN
	bInitFB := FALSE;
	//Fehlerstruktur vorausfüllen
	stError.ObjectId := nObjectID;
	stError.HardwareGrp := E_HardwareGrp.Nothing;
	stError.POU := E_POU.POU_FB_CustomUnitType1;
END_IF

CASE eCurrentState OF
	E_MachineState.MACHINESTATE_Active:
	//BasicActions ausführen
	IF bSuckOff THEN
		A_SuckOff();
		IF nStateA_SuckOff >= 80 THEN
			IF nStateA_SuckOff >= 99 THEN
				bError := TRUE;	
			END_IF
			bSuckOff := FALSE;
			nStateA_SuckOff := 0;
		END_IF
	END_IF
	
	IF NOT bSuckOff THEN
		bBusy := FALSE;
		eCurrentState := E_MachineState.MACHINESTATE_Idle;
	END_IF
	
	E_MachineState.MACHINESTATE_Reset:
		bError := FALSE;
		
END_CASE

IF bError THEN
	eCurrentState := E_MachineState.MACHINESTATE_Error;
	bBusy := FALSE;
	aPumps[nPumpNrWaste].M_Off();
END_IF

//Prozessdaten aktualisieren
stProcessData.nObjId := nObjectID;
stProcessData.n32Data[0] := BOOL_TO_DINT(bIsInit);
stProcessData.n32Data[1] := eCurrentState;
stProcessData.n32Data[2] := stError.ErrorId;

IF aValves[nValveNrSlot1].bDigiOut1 THEN
	stProcessData.n32Data[3] := 1;
ELSIF aValves[nValveNrSlot2].bDigiOut1 THEN
	stProcessData.n32Data[3] := 2;
ELSE
	stProcessData.n32Data[3] := 0;
END_IF

aObjProcData[nNotifyId] := stProcessData;

ACTION A_SuckOff:
//entsprechendes Ventil und die Pumpe gleichzeitig einschalten
//wenn Action zu Ende oder ausgeschalten wird, wird das Ventil zeitverzögert ausgeschalten, damit
//sich das Vakuum erst abbauen kann.
CASE nStateA_SuckOff OF
	0:	//Ventil und Pumpe einschalten
		IF bSuckOff_On THEN
			IF nSuckOffChannel = 1 THEN
				aValves[nValveNrSlot1].M_On(1);
				aValves[nValveNrSlot2].M_Off();
			ELSE
				aValves[nValveNrSlot2].M_On(1);
				aValves[nValveNrSlot1].M_Off();
			END_IF
			aPumps[nPumpNrWaste].M_On();
			IF tTime > T#0S THEN
				nStateA_SuckOff := 1;
			ELSE
				nStateA_SuckOff := 80;
			END_IF
		ELSE
			nStateA_SuckOff := 2;
		END_IF
		tmrTime(IN:= FALSE);
		tmrDelayValveOff(IN:= FALSE);
	
	1:	//Time
		tmrTime(IN:= TRUE, PT:= tTime);
		IF tmrTime.Q THEN
			nStateA_SuckOff := 2;
		END_IF
	
	2:	//Ausschalten
		aPumps[nPumpNrWaste].M_Off();
		tmrDelayValveOff(IN:= TRUE, PT:= tDelayValveOff);
		IF tmrDelayValveOff.Q THEN
			aValves[nValveNrSlot1].M_Off();
			aValves[nValveNrSlot2].M_Off();
			nStateA_SuckOff := 80;
		END_IF
		
	70:	//Abbrechen
		aPumps[nPumpNrWaste].M_Off();
		nStateA_SuckOff := 80;
		
END_CASE
END_ACTION

METHOD FB_init : BOOL
VAR_INPUT
	bInitRetains : BOOL; // if TRUE, the retain variables are initialized (warm start / cold start)
	bInCopyCode : BOOL;  // if TRUE, the instance afterwards gets moved into the copy code (online change)
END_VAR
eObjectType := E_ObjectType.OBJECTTYPE_CustomUnitType1;
eObjectGroup := E_ObjectGroup.OBJECTGROUP_Target OR E_ObjectGroup.OBJECTGROUP_Device;
END_METHOD

METHOD M_AddChild : ERRORID
VAR_INPUT
	pObject : POINTER TO FB_Object;
	nSlotNr	: UINT;
	nIndex 	: INT;	
END_VAR

VAR
	pSlot : POINTER TO FB_Slot;
END_VAR
//In den abgeleiteten Tool-FBs wird überprüft, ob das entsprechende Objekt als Child tauglich ist
IF pObject > 0 THEN
	IF nSlotNr > 0 THEN
		pSlot := fbSlotList.M_GetAtNr(nSlotNr);
		IF pSlot > 0 THEN
			IF pSlot^.P_pChild = 0 THEN
				//Object darf selber noch an keinem Parent hängen
				IF pObject^.P_pParentObject = 0 THEN
					pSlot^.P_pChild := pObject;
					pObject^.P_pObjCollectNode := pObjCollectNode^.nodes.M_AddNewNode(pObject,nIndex);
					pObject^.M_UpdateParent();
				ELSE
					M_AddChild := E_ErrorIdObjMgmt.ERRORID_ObjectAlreadyOnAnotherParent;
				END_IF
			ELSE //Slot bereits belegt
				M_AddChild := E_ErrorIdObjMgmt.ERRORID_SlotIsAlreadyOccupied;
			END_IF		
		ELSE
			M_AddChild := E_ErrorIdObjMgmt.ERRORID_InvalidSlotNumber;			
		END_IF	
	ELSE
		M_AddChild := SUPER^.M_AddChild(pObject,nSlotNr,nIndex);
	END_IF
ELSE
	M_AddChild := E_ErrorIdObjMgmt.ERRORID_InvalidParentObject;
END_IF
END_METHOD

METHOD M_CancelAction
VAR_INPUT
	eAction : E_Action;
END_VAR
IF eAction = E_Action.ACTION_SuckOff THEN
	IF bSuckOff AND nStateA_SuckOff < 70 THEN
		nStateA_SuckOff := 70;
	END_IF
END_IF
END_METHOD

METHOD M_CheckAction : ERRORID
VAR_INPUT
	refActionData 	: REFERENCE TO ST_ActionData;
	pCorrelObject	: POINTER TO FB_Object;
END_VAR
IF refActionData.eAction = E_Action.ACTION_SuckOff THEN
	//BottleState prüfen
	M_CheckAction := M_CheckBottles();
ELSE
	M_CheckAction := SUPER^.M_CheckAction(refActionData,pCorrelObject);
END_IF
END_METHOD

METHOD M_CheckBottles : ERRORID
VAR_INPUT
END_VAR
//Wastebottle OK?
IF nBottleNrWaste > 0 THEN
	IF NOT aSensWasteBottle[nBottleNrWaste] THEN //Voll
		M_CheckBottles := E_ErrorIdCmd.ERRORID_WasteBottleFull;
		RETURN;
	END_IF
END_IF
END_METHOD

METHOD M_CheckProcDataType : BOOL
VAR_INPUT
	eProcDataType : E_ProcDataType;
END_VAR
END_METHOD

METHOD M_ClearAllProps
VAR_INPUT
	bIgnoreParent : BOOL; //Es wird das gesamte OD gelöscht. -> Zeiger auf Parent nicht mehr gültig!
END_VAR
fbSlotList.M_Reset();
SUPER^.M_ClearAllProps(bIgnoreParent);
END_METHOD

METHOD M_ExeAction : ERRORID
VAR_INPUT
	refActionData : REFERENCE TO ST_ActionData;	
END_VAR
IF refActionData.eAction = E_Action.ACTION_Init THEN
	bIsInit := TRUE;
	RETURN;
ELSIF refActionData.eAction = E_Action.ACTION_SuckOff THEN
	IF NOT aSensWasteBottle[nBottleNrWaste] THEN
		M_ExeAction := E_ErrorIdCmd.ERRORID_WasteBottleFull;
		RETURN;
	END_IF
	
	nSuckOffChannel :=  DINT_TO_USINT(refActionData.aParams[1]);
	IF nSuckOffChannel < 1 OR nSuckOffChannel > 2 THEN
		M_ExeAction := E_ErrorIdCmd.ERRORID_InvalidSuckOffChannel;
		RETURN;
	END_IF
	
	nStateA_SuckOff := 0;
	bSuckOff_On := DINT_TO_BOOL(refActionData.aParams[2]);
	tTime := DINT_TO_TIME(refActionData.aParams[3]);
	tDelayValveOff := DINT_TO_TIME(refActionData.aParams[4]);
	bSuckOff := TRUE;
	
ELSE
	M_ExeAction := E_ErrorIdCmd.ERRORID_InvalidAction;
	RETURN;
END_IF
bBusy := TRUE;
eCurrentState:= E_MachineState.MACHINESTATE_Active;
END_METHOD

METHOD M_GetAbsPos : ST_3DPoint
VAR_INPUT
	pChildPos	: POINTER TO ST_3DPoint;
	eTargetRef 	: E_TargetRef;
	nParam1		: UINT;
 	nParam2		: UINT;
	nParam3		: USINT;
	nParam4		: USINT;
	nZLevel		: USINT;
END_VAR
VAR_OUTPUT
	nErrorId 	: ERRORID;
	lrAngle		: LREAL;
END_VAR
VAR
	stLocPos : ST_3DPoint;
	pSlot : POINTER TO FB_Slot;
END_VAR
IF eTargetRef = E_TargetRef.TARGETREF_Slot THEN
	//Slotnummer checken
	pSlot := M_GetSlot(nParam1);
	IF pSlot > 0 THEN
		stLocPos := F_Add3DPoints(pSlot^.P_stRelPos,stRelPos);
		stLocPos.Z := stLocPos.Z + stDimension.Height;
		//kann es mal sein, dass hier das ParentTarget = 0 ist?
		//ja -> bei der Workplate
		IF pChildPos > 0 THEN
			stLocPos := F_Add3DPoints(stLocPos,pChildPos^);
		END_IF
		IF pParentTarget > 0 THEN
			IF pParentSlot > 0 THEN
				M_GetAbsPos := pParentTarget^.M_GetAbsPos(pChildPos := ADR(stLocPos), eTargetRef:= E_TargetRef.TARGETREF_Slot,
															nParam1:= pParentSlot^.P_nNr,
															nParam2:= 0, nParam3:= 0, nParam4:= 0, nZLevel:= 0, lrAngle=> lrAngle,
															nErrorId=> nErrorId);		
			ELSE
				M_GetAbsPos := pParentTarget^.M_GetAbsPos(pChildPos := ADR(stLocPos), eTargetRef:= E_TargetRef.TARGETREF_LeftBottom,
																nParam1:= 0,
																nParam2:= 0, nParam3:= 0,nParam4:= 0, nZLevel:= 0,
																lrAngle => lrAngle, nErrorId=> nErrorId);
			END_IF
		ELSE
			M_GetAbsPos := stLocPos;
		END_IF		
	ELSE
		nErrorId := E_ErrorIdCmd.ERRORID_InvalidTargetSlot;
	END_IF
	
ELSE
	M_GetAbsPos := SUPER^.M_GetAbsPos(pChildPos := pChildPos, eTargetRef:= eTargetRef,
													nParam1:= nParam1,
													nParam2:= nParam2, nParam3:= nParam3, nParam4:= 0, nZLevel:= nZLevel,
													lrAngle => lrAngle, nErrorId=> nErrorId);	
END_IF
END_METHOD

METHOD M_GetActionBusy : BOOL
VAR_INPUT
	eAction : E_Action;
END_VAR
IF eAction = E_Action.ACTION_SuckOff THEN
	M_GetActionBusy := bSuckOff;
END_IF
END_METHOD

METHOD M_GetAllProps : ERRORID
VAR_INPUT
	refCmdData : REFERENCE TO  ST_CmdData;
END_VAR

VAR
	i : UINT;
	pSlot		: POINTER TO FB_DimSlot;
END_VAR
SUPER^.M_GetAllProps(refCmdData); 

nCurrentPropIndex := nCurrentPropIndex + 1;

refCmdData.n32Data[nCurrentPropIndex] := fbSlotList.P_nCount;

fbSlotList.M_SetCurrentToHead();

